(* CoDeSys 2.3 project: cy-wg-017-002.pro *)
(* Title: cy-wg-06 - ClevergyAS *)
(* Author: Andrea Ravasio *)
(* Libraries: Standard.lib 2.12.10 13:48:34, Util.lib 26.9.14 09:12:46, Visual.lib 2.12.10 13:48:34, WagoLibIdent.lib 25.2.13 10:12:16, WagoLibStatus.lib 2.12.10 13:48:32, SysLibFile.lib 2.12.10 13:48:34, SysLibRtc.lib 2.12.10 13:48:32, SysLibSockets.lib 10.2.11 08:20:54, SysLibEvent.lib 2.12.10 13:48:34, SysLibPlcCtrl.lib 2.12.10 13:48:32, SysLibCallback.lib 2.12.10 13:48:32, mod_com.lib 2.12.10 13:48:32, SerComm.lib 31.5.11 07:54:36, Serial_Interface_01.lib 22.4.13 11:50:14, Modb_l05.lib 13.5.15 09:30:08, Ethernet.lib 2.12.10 13:48:32, MBus_03.lib 9.2.13 16:51:58, WagoLibModbus_IP_01.lib 24.7.13 14:05:58, WagoLibMBX_01.lib 20.3.12 15:32:40, LON_01.lib 28.9.12 13:05:10 *)

(* PLC configuration (modules and I/O channels)
VPN_ST2 AT %IX30.0 [BOOLOnX_I] Ch_1 Digital input
LAMP_AL AT %QX18.0 [BOOLOnX_Q] Ch_1 Digital output
KEY_QE_ST AT %IX30.1 [BOOLOnX_I] Ch_2 Digital input
CIR02_EN AT %QX18.1 [BOOLOnX_Q] Ch_2 Digital output
CTL01_ST AT %IX30.2 [BOOLOnX_I] Ch_3 Digital input
CIR01_EN AT %QX18.2 [BOOLOnX_Q] Ch_3 Digital output
CTL02_ST AT %IX30.3 [BOOLOnX_I] Ch_4 Digital input
AT %QX18.3 [BOOLOnX_Q] Ch_4 Digital output
CIRD01_A_AL AT %IX30.4 [BOOLOnX_I] Ch_5 Digital input
AT %QX18.4 [BOOLOnX_Q] Ch_5 Digital output
CIRD01_A_AUTO AT %IX30.5 [BOOLOnX_I] Ch_6 Digital input
AT %QX18.5 [BOOLOnX_Q] Ch_6 Digital output
CIRD01_B_AL AT %IX30.6 [BOOLOnX_I] Ch_7 Digital input
AT %QX18.6 [BOOLOnX_Q] Ch_7 Digital output
CIRD01_B_AUTO AT %IX30.7 [BOOLOnX_I] Ch_8 Digital input
AT %QX18.7 [BOOLOnX_Q] Ch_8 Digital output
CIRD02_A_AL AT %IX30.8 [BOOLOnX_I] I 1: Digital Input
CIR03_AL AT %IX30.9 [BOOLOnX_I] I 2: Digital Input
CIRD02_A_AUTO AT %IX30.10 [BOOLOnX_I] I 3: Digital Input
CIR03_AUTO AT %IX30.11 [BOOLOnX_I] I 4: Digital Input
CIRD02_B_AL AT %IX30.12 [BOOLOnX_I] I 5: Digital Input
CIR02_AL AT %IX30.13 [BOOLOnX_I] I 6: Digital Input
CIRD02_B_AUTO AT %IX30.14 [BOOLOnX_I] I 7: Digital Input
CIR02_ST AT %IX30.15 [BOOLOnX_I] I 8: Digital Input
CIR02_AUTO AT %IX31.0 [BOOLOnX_I] I 1: Digital Input
CIR01_ST AT %IX31.1 [BOOLOnX_I] I 2: Digital Input
CIR01_AL AT %IX31.2 [BOOLOnX_I] I 3: Digital Input
CIR01_AUTO AT %IX31.3 [BOOLOnX_I] I 4: Digital Input
0750-0478 2 AI 0-10V 16 Bit S.E. [Type_8_2_Channels] node 3, in %IB56 out %QB36 {INTTypePAAssignment = PLC; INTTypeModule = plugged}
  VRD04_ST AT %IW0 [WORDOnW_I] I 1: Analog Input
  VRD05_ST AT %IW1 [WORDOnW_I] I 2: Analog Input
0753-0648 LON-FTT [Type_55_1_Channels] node 4, in %IB4 out %QB0 {INTTypePAAssignment = PLC; INTTypeModule = plugged; DataStream = 1F8B0800000000000400ED5D7B6FDACAB6FFFF4AF73BF820DDA3560A0D06421E27CD1605A7419B470E9074576D851C3310EF1A9BE347D29C4F7FD79AB18D8DC70F02348158DAEA26F678CD5A336B7EEB31CBE3F33F7ECD34E18198966AE81F0BE287524120BA628C557DFAB1E0D893A2582BFC71F1BFFF73DE36F4966E1373; DataStream = 222B44808774EBEC97A57E2CDCDBF6FCECF0F0F1F1F1C363E583614E0FCBA59278F857A73D50EEC94C2EAABA65CBBA420AFE53E3F4A70AC2B5694C4D79D682C6A7A5B352E9EC18FE3D3A2B8967A5DA59A90A3F0AC25FEAA42BCFC8C7C217796A8C6E55DBB04D4357954A09C418106DD234146746745BB641BC8631C3DF1F0B; DataStream = F5F15878321C5350D815E19E98C05E9738F0F4A56ACE1E6593DCFA63724A3B1AC80FE45AB6EF3F161A67DF3FABF677E5A958128F8B8F53E15D935844FFAFAC1BC227792ADBB62CD44BE2A7F7DFDBBDEE48278F05A1638C1D8D749DD91D3181620106541070483BB2F9B377F737516C8B5E5BBEEA5E84CB43329B6BB24D5A63; DataStream = E0589DA8C4F4EFC15D1CADD6F8A2541278FF9D1FBAF7034F0C14634E2EE016FB11B8F32779C2EBF8BFC0D5963E26BF2EC4F343F6C3E7EB3081319F699CA58BC1E5F55037C68449B67890DEF41FE1360D37E999EA54D5658DDB3474D37FA465B50DE527195FD8A6434006EFCF40838EAC8F65DB309FFC368B2B8166BD39EA92; DataStream = AC5D4C64CDA2CDFC2B7EAB0EC18966D38D4319FADB6F256904B5AF6138A082B096CE7455FB58C0CE0BC261604088FD68983F6F655395EF3462052765E95EE0569AC63C4F6B9235C7D79ED3F2B2FA0454086F867528558F38BAD4BD1D8E8CBBBF4726F98F43AC386D5A6894FEA0F6BDA6D12621A50936E56A53268D5A41ABB2; DataStream = 6B5654BBC418EDA22DB3691823AAEA03A28F87EA8C4E6DF0CF703BF957A85DE0CFE5767DA210F581049A06AF2C097F6DAA86A9DA4F0BE1FD2BA19603623EA80A193E81E6D5959FBAF1A891F1948C411B0377428F345513900106F2A2A5CF1D98D4C58530CB60F526AA827373D1357460227825D4B461E81375EA98D4AEC02A; DataStream = 9913D35689B53CA82DCBEF6A495996AF871EFBF4649381FA5F7251393FF47F0756FD61FCB27FB58850494284CA261101BC0DDBB132008231705BA6E281DFF2D5C341398783EC70D073ECDDC283DADEE0C171121E1C6F0C0F26AA46D045C8E21E5C42DB3E364D770FFCA61BC4035FD1D301C12399010F8E723CD85FF7402CEF; DataStream = 0F1E5493F0A0BA513CC8EE20E03A47D39FC54558B47DF5A050CB41618F9D84F2F1DEA0C269240DC54688450DA58DA2C2DCC80209D4F45F1B59828645D3570F08C73920ECAF97B06AD010B9B3C838A6B27C7EC8CB5E3F2FA59D9CA02E8A3119EAE28A296ABA286F55D376644D9838BAC2568B70A7C1A02E679E574A2327ACD5; DataStream = 3C8F9C0DFF5F5F1E199A67CD234769673004BE366CD012AC92408AD332DA323705C26BF30D7DF1F28C321BA197CB2843EB8C19E508E51C18F60B185EDE475C1117F627B37C9294493AD95826C906D5C2E53B9B67C10554C401C9E8320449E7C0B05FC0B07B1EC3FE64934E4E9290E16453C8206BB239CB020A75D6300B24B8; DataStream = 347334D82F34D83937A17C9AA3C136D120B38F9003C25E02C2EEB907FB8408491985938D651430E62799F28CDAD380B5CD82082ED91C11F60B1176CF45D81B3C104B492E02BDBB1944B87F9095D1CC18674285AB46431CC12C67CF2704C8E7E8B05FE8B07BFE8298C3C3EF81871C1BDE3836EC9CE7B04FD07094080D471BDB; DataStream = 85802BA34C3B101417B059F66D0897768E0BFB850BBBE733EC5348F17A81214785B78C0A3BE72DE4A0B06D501838F3790E0C6F1D187277214F31B883B40087729E81CCE16147E1619FD20CAF1A1E726C78E3D8B07331C53E41C36B8C29CA790632C7855DF419F629A478BDC090A3C25B46859DF3167250D83628E419C81C18; DataStream = 7277214F31F883B400874A9E81CCE16147E1619FD20CAF1A1E726C78E3D8B07331C53E41C36B8C292A790632C7855DF419F629A478BDC090A3C25B46859DF3167250D83628E419C81C187277214F31F883E48243F3EA4B9E80CCD16147D121CF326CD16F4068A82B76EE35BC755CC8C3891C16C2B000DEC2B5A1EA79F2F14D; DataStream = E3C2EEF90B39306C1918F24D891C17727FE1E560E13409154E37060AD6A36A2BF75940A171D9446F41D27194321E00E912CF6161BF60217717725C08E1C2E71C17725CC8DD857C4FC21BA4B0CF90173EE6E0B0834E43BE27B1C51C034243BE21F1D64121F718724C88B80BF986C49BC785DD73167260D83E30E4FEC25BC785; DataStream = DC5FC8138F1E287CEA35F20D891C16727741C8714158C2857C4322C785DC5DC83724FC410AFB0CF986440E0E3BE834E41B125BCC312034E40986B70E0AB9C7906342C45DC83724DE3C2EEC9EB39003C3F68121F717DE3A2EECBDBF10B9632D6EA5F17C7ED836F48E6CFEECDDFD0DACD1AB4BD7AC8BF37F7C6B34EBC3FAB7F3; DataStream = 3F7ECD34E181981650FB58103F940A02D11518307DFAB1E0D893A2582BFC7171DE906D5933A617E797AA46849605FFB38949C6F0484168C2CD5B9F44156960339CC28F05FC17FE36CC996CFB8D6AD8A623FF6D9881E70AC2B56CDF7F2C34CEBE236A99F28C92B18477BF4E6AEFBF83085F6048ACEF48D1FA3E18D6BBCD7ABF; DataStream = F961F8F51A9EA430F7B110838305A14F26C0AFAE90C456A8D2035B9ECD819FF2A158392C97C4B2209E9C954B6762B970B18CD69415EE55E1936CB923308095AAD8DF6A3F0A025DC2207E41A0E0F9B1705C2908084B1F0B74604DF21F8758365C7BB0D9C3886320A1341A0CFB378D2193148606465355D89314EB26F0F8081E; DataStream = 2F08A865C87E41B8D155E8EC9F9AFDAF96FE206BEA58B06C132616BAB10CC754C83FA7F6BFF84205D89774672678E491BB918D73F74B9D39332A0A800CFB5D143D61FAF17248DD9B0E4F0A5FF4813AD55DC57245F12499048648D0E129AB202077842D0677488F10145364BAD12DDA0BE8D414E6C26AE936991293F6D5B206; DataStream = 8AACC9EC8F859C474795234F3CDA134FB89BEEA0F5B92B3547ED5EF77341E84D2616B129A1A8C02A23829D917A40DC72485CB7D5B62572215DB06101180E77E26264ABF02793921BF9E4E2A59CA99AA65A4431F4B195494E98E96F95C55AF2175013B402AC3C6A82208FC7A0E3165F8C56AFBB60FF88C7FE18B5DCA7C1183E; DataStream = F218F670C8EF24E3FA2F2F782E7B3CD71909C1C6C700786DF32969ED27328DECD81EB7158F5B5E0F597569706F20C52CCA54A90470A05289C8478D40824E0DAE7AFD340119918826F9F07052BC536DC171991700F19883B4DD95131E60754564A83D0B19C45A9CA8CB8E0375A39E639F5CD3E2DCE9C42EEAC69824ADA94CFA; DataStream = 69E9F14BC9E2F4B3052D15034A2AEE928E7E526D7F72960472C1CF98C9AACE63FF536B7899A26F63F7E178B6FD89624D57B64AC2B14045807F0236D115E8382850F9D813A90BCAF04C8174FA68BC3854CF741A69AD2244352244D517A21A14226056016F05059BA48B72CCB7A4D42624C842C5108C89804D5592CD883E5BA2; DataStream = A129EB964C431EEA2C98E9729D7017CAAF91FB78BC68B4018C1E4CD6AA60BE0228948F8EC270B70A089C7291CE25132F196B1154C13580FBF847702931163E9B86335F1BB2A7F378C89E867A581BC0D25038AC52CFC2DE3BC3D088AC6F03B66A0B15823E9FC9BF451FCD00C26CE859F3376F3A181F37BA6341DB894AB4F133; DataStream = 457128892451D222E9DC94E4A62404C06B5B9229A3B29E4AF24DCB730CCEF35C6E17E01DFB1EF7041416A11B5CC4891B1CB1C48D7881E4C848449FD531FF39B27939EE55A5E2E685E6406C05A9D6701CAA3F822BD4CB4856431949CB966D27D183484A487A4FBBF1EBF1E67392AC87504A5214B939C941AC247129C905F789; DataStream = 1949D62C3E2159DB7E12A2EB2337721493F7CA9E9A648660644C462EB9F854846B90B62DE0806844B1A985D792A3F40CD949CB253662C4369681C5CC644296EFB9D948796CFA9C6D2CABEF42404C225531D5B96D700D72A6C0611C20B169CEEBA6293F7D136B3F50DD2FD90C4D0C41C6CB02615BA50B8F17B75A2CFA4800AF; DataStream = FDA77802D6FBFDFAD714F928F430022E22D43CF1181FC09A5813947BD9040787981992C4747534E0818CB607C1348072E5938870CB43C2994BB6641A57F5FE42E032D7D6FA127F138F7E2CAD99387464C9AEFAA0D16A2D86E2F9468BF6F36F471E6774C6C4EA71F5A452AB1EA7C566EE30FCFBA6DE0C0C0317193931DA92F4; DataStream = 55DF483FD92B79D0CF44C6615ADA320C88E55542E7CC6B76A38E482A6866DE0E096CDF9C6E167E18FAB0D059683563D0870B3EFE43CF051F16488FD4B1275B147B6A02D3BEEDC638B1E2AFEBD8FB127E8B604DB66CFA6F0A6E6A4B23A1117D6ADFAF1F02B8F27BE4E20740EA0A62F5B4745214BDF48AF7CCABCB946241C266; DataStream = 52A59B8FE3D2371D62A5E23A98ABEE3FAC12A1AF01B362608B4F5CD4A09C54822112111EC0394EF6FD62423E0C840867B3125D68F5411D3BB226E082A5EB74033963C62E522CC5A78EA2BCC203A5CDE40CE2139329FC8A2BF22B6E87DF72567ECB2BF25BDE0EBF95ACFC5656E4B7B21D7EAB59F9ADAEC86F753BFC1E65E5F7; DataStream = 68457E8FB6C36F2D2BBFB515F9AD6D87DFE3ACFC1EAFC8EFF106F9CDC6E1497AB29EEBDAC0B3272F0CBEA7CF67FDF48571584C307469BC8B5B327A9941594CB07AA9CC6FC90266466831C104A632BF25739819AEC5047B98CAFC966C6366EC16138C632AF35B329499815C4CB094A9CC67B69A1BABFAF322023F0B8305F1B8; DataStream = C131E3EE65A6C403B8E93A721F66DCFB1B404F44360F8499A1DBF707C2587E3A10EE0D07AFA8BA63930381150467CC9A66CF9C554A58E5CFD91CFA4A647EC413CCA145C57CA28F25A503CB4189574907AE14BF7A6274704057895FB941F98C5189D73DDA604BC254168932995B0C1D270A37121FCB89150F707B4B6294FDA0; DataStream = FA0A147B1539AA3C39EE29917841F0FE9624393AF5B58B2ECEB56B64672E9904FDA22DB62ECF8081CC0AF2700B875CAC4ACA61055E6F58277F13C8938B8B1DFB137FEBA70EC2CE9EBF658F6335F3816B2B19F3B6E1D67FAC9030F79E49C8974705D2FC875E36471E27F09A6BC8136FB504390ABC767EFC99FB54ECD5C3986D; DataStream = 8F55DE8E302821B6FD11BB61C51A65DEBBA7F52454FD47B815162A27A994431E4325BCD8EC98ED3756539258B7B6E82F691355F6BB89AF3039CE2AE2DC2D541A69E4816859AA66FCD226FA44BAA4DC32B670B749D2CE43DDC54B7CF29B5EF243A0E8DEAE524FC3DDD0A27A38B28D11E26C92DEAA8B4E0545762C045B179653; DataStream = E565385BA5387B8B29F61890ADF240F696ED9DA5EE48F2B771DC9DB7A51D701F6AABBF056AB932AFB095C3055A2A192D934908C57E2FACB22026396E89D34E2EA272A2981D085D442EA8EE66EC227261730783177EF1D08E462FFC12A01D0E5FCAFC3DF895E2974DA3D9E9696086FC57C157A968E206FEB320AD8DBD7D1E34; DataStream = B1CCFFD3D41978D82B18DAC06319CC2DBF5C8B798E2E8D9735BA09A3B0825E26F8C794F47A06788D903B5CCEEB3A9FA7BEF9A5B59673C352E3E2D32C45F2F07C244A9DE3E967C43CF0EA79B65F1CD927F2F8F00BF8DE2810ED3CB55492F38AD1E3686EA764447D4DA5D5D538758BF714B77FCC852F64865AAD30CE70F37220; DataStream = 706C95960F328BF7AA1635A11BD749DF917203EDE71F2503B1F328701A4BE8388956F3C0A7FC8A1206BF314BE012E69D8553AE7243E8F4090987D05C231DEE3629843642DDC587D018A9AEA98881CDA3F262F7E8B4B224F9B31392A889E157886A4145745FBC9968F234BB99DB1B6D4C2DD67073B6C556930E51FA462457F1; DataStream = 544685CFFB06B652C56C4278EABC0149166BE8F7977234550B898CD79163ECD27891728E9E63178D49917A65D63A52188E8D2F9831422F52DCD19B13BDA8A8A6E2A86BE9950174462E9D1729F470E7C46227276E60525C4A2F52F8D121CABDACABD07171223BDA5A3333F3698D28AD172906B924647C272B3F411C5573CCB5; DataStream = E667E2D21AB9B47E53D95FEF81984553D6A75999E786E4065019512A2F62496EC0AE6E400A07C96C538C140B22E1BBABE6CAEB832B0BF1696D737DA458941BFACDA0A26D146744B6B22F9098D94162B8D3E2127B11CBD230663347778F3AB0565CF85CB914A0B885459FDDC65C42DF640C36469B14EDEC8E18571894638494; DataStream = 46F6D6FCB0B4F2424F8EA2AA17E7C8211E3EB4864CBE3823551F79045FC4DEB093888B60CAD79147A35446FCC33BB761633AB2EE00A629866E9B869691756E4E6646298D5C4A2F14B5CCC127635BF76B4802AAE4D5E4FC7E43C36440A36DAAE3ACE015278647E6452C4C9FCC0DD32ECE64EBE73A629894CC08C9BC8855F138; DataStream = 52F56911BF8EB58E2CF3052DFAA5AD17B1294181D0266C4A20A4F52256856E861475C356274FC5F16AA13E572AB605C2088EB61BF7A758953EB1F8EFFB665A38700FF07836D748F2CEE9338EE83B1182A6C52F85C43ECD0732CEF0DA06778B2DF0FC364EDF5A23D1BF78079B7E40F3196955CB7D7029FF484B5D5856956C65; DataStream = D77051B6125B6DB4BC43185F6AE44E8AF78EC42796715F9AA0FFA34722399AE695AFA5EAD5609D3385C3874D259D35B25CFF1177FC54CA6123BEA0B42D3DDF6ECDF355DCF4B8B7457094B1F0A57C5C0B9D47533EAE88FED6227EB105F71E68ECB2F23B16814FB98407C39BF672D26B1763029E38B18406D12CD5C9B2C54877; DataStream = 79E82728EDC0409C8414993BE757B7F586308B394020EE8CB1F0072F93A6D8279FB0A5538D9D7DEBE23CD03EFC97B0F872C2509EBA67FD2C36B82ECE59655D28212FB84B382AD1657FD4BD691784BEFC48DBB0213A0C53192075DD56654D901505632F93E0DE35975CEF5AEA8E86BDD140EA3633507AC4FDDD14527DA921B5; DataStream = 6EA5209751261B9A611141D601DCE507E21E3DC625DB68F706D2E8B2D50E512C27501C13B485E9349B525B1A46495722A4FBF4C84E60734C3F4963984FDEF704B8D49B2D188261AFFF15D65DEFCF9BEB20F16A9438B06CCC569CAA51BF1EA47A94427585695BA2CC0ED83B0C683457BD6B41F5F6CF0D5C55BB0719B49B9685; DataStream = D878BCE9849882E55001C10CC510FCEB520211FF8C9069FA33A919C64F3CF2378D129B4B4A2B49B125D3344C014FE19C131DBD9658351CB0A1BFACB7DAC99AED931C2F319DCCA9D4EF27AB757828555D58E456E2C7F2A6DB94FA5FB08E2A49A97D96519F61140E51035346A3D55B6639AAD66196F125C8B140F3285C8AC356; DataStream = 47EADD0C97C9D62264BFA8B05A1E058BE29D420482ECC710FDD2EA367B5F96691E47682E1DCAEA2718B944EB37C3AB65922751926C35334365D8A0B3730C9B091F31806AA3210D063065F5DB25253B4D018C3BF26400924A3DEEA908407A20497F8E5ADDDB7A1BB7ED030BA2149D33B7F5977A8BEB7586EF074889D9B0E7D8; DataStream = C59ED03B2661166EE663F4E1FCF9BD07AD24DC09AEB74757521D543C0C43D1C5B34C726218762CC9CB5E6FB84C32BACE9BE4CE99D2E305F1835E28E13B9C655967AF29BC8F21DE943EDD7C0ED38EC2522B40D561AC6722DEEA5EF6C2B4A3133C78B2C0875C9DF1C1D7C150EA44BB88AECFE1BD7BB6B4A05A825B6B10431434; DataStream = F246E26966318A2621B232B8F83A982EDD3D44299B0C8D5E17BF961652DC62140FB1A731A15BC8D095319968AACEC50220D9BBBC6CB7BA2197A418D53F561C8AC5B52A9B541DBFF407233F939F60F90A6368691B54AAC08689074302A0F3BD6C8E1F65DC3B61D7E244BCE9FED9ED7DE986F8892AAF67DD03EF54B9C3282F71; DataStream = 4A916B4E14FC84E538AED37447A06B08CB94E79859D0B9D60049F670B69AAD213D16767939EB3E4B2B92ADB73B41BA49BEC1D0B065EDD0AB25A085A00FE85BD3FE44E11DA6710C1DBAA2156660EC2DC16B0CF38567D0D94497016DE2466DD81B8E06B70DCA9398EC5424F2C2DD205FA25F4E762E12E973B74596E857923D0C; DataStream = B7381AACB65B20CD264D23B22970437E20DF06BBDDEE0CC1FDEF8787270A0D49E4E3462748BE9CEC7030F2F7EAF47E05F6AF5A9FAFF8FC73BC8FA40EE2040875504EF145B8039436F211C58C3A227CC269631ED1488E9D8A1993D4E18E30CDB1AF31B453473ACA7774A95E02122C83529CA3D1EA23C910419EE30F0401D58A; DataStream = D9895EF7A508E1E8A244C24593E0B786C7E0A61BCE1DB8EBEF68FDC3FB4CDD0CFB9F42B82FF24280401FE00123C25806FD7E8707D8EFC887E987033032A6AAFFD420504004B7124C1C763DB8B9BE0D751D5DB561F170879BBAE2D94771280D8691618C2EDE987E569B31DA176FDAA26B39D4DF8CA5E204A23FA8A6A1E3FB26; DataStream = 80DB689A886E312782BD400CA19D72CF8F3D5C16A4EE6DA3D7B91E75EA7F8538882EFA1007F29D8E8EA4065663EED89984EDF4BAAD61AF4F0D71C8EE71C291B0B0BE4D856924669C91A77DD45B5D9C3DA91FF2F6CA9C1C057ED15790E773CD73BB62034AA45D1FC2BF10FCF5C2F17A94F51E449426A3953A2A517A513E193D; DataStream = F00169A2228DE2977ABFDBEA86228D4A395B8876E286689177E457CC105D67C97FB68D472CA2612B65BEF48E3D97665BBA95DAA3E878FBB7B826227837C9EBF3DB718D41F06E92BF7605A6E559625592FDB4B63A21C2409E102046ED02B56496F0EE53BD818703FB871494B9E079BDE489446DC235FB8EF653A64E2A719D94; DataStream = 93DD354A74103006CC1E47E857E3E85792FD354A7FC80CDAE125AD0D7CD754ADB9263FBD8FF67214D74B35D969A3BD5C033C51EE0F04BA2DD1C0CC9902782241483047388E13AE16D76D2DD995A3DDC4CDC8491CD19364372E8EF7FEB07BC074007E250DA2588A55B8528AA347FBA6E4358605DE72E175133B6A628DE3F3A5; DataStream = 421DB243B12EF232D38A58D7FF7706AC93684DA6FBE214DDFC30C9CC78802B7E51109F72AFDFA9B73959712B402FE6D9666B50FFD4969AC9A8C70A833CCEBC378DB8046FAE9BF521EEACD78737836414BC262626997CB25EA9610CE581D4BEA48E503206BAB93C3974C45312ABF576BDDF49863D577EF73D2A3C2A88153771; DataStream = C9F6A5EB5E7F081EC6E0CF649CEB7925638933D4BB05EBDF6A4AC99816D29D184A5217A73A19B5FAAEC6B1294951BC7EE796CB5E14951A3454CDA23F8DB654EF73D4270A4A219A6EF95F02C9C83473B0C61D45A63BB49A48F54EC7E252A63461FD0D5B975FDDE16D727086B72A9FD70777B9723699424832A1F926ACF514FC; DataStream = 5A4F6E579D7AF706D3A0C37E386E8B2EB268070855B4B222A983BED4E9C18A8B74C0D973621D04AAD5B04285A6F598181375EAB8603D674E09FD0E23B7DBEB7EEF73BF1E9EFCE87264FA446BB08A5E0D16AD4913DE850BB3B836C6D7B3BE3490C25B1F9CD5FA8B280E50679DF9DB0E2061E2028E928E2E60260540A02C68C6; DataStream = 3491D3762FE4FF7362C9B62143CC7AEFCFC322D58B3B8C83C6F5106FB06F8EC574D5EED59BDC09E0EC5A393AED4C714C13BC0B0D7746E531F4E5F6FE41684D42DC3CCA96702F6B2CF643FDD69E0EA0816A098FAA8631AD05165D301D9DEDDD9AC68C3D8EAFED63EA7EF1FC87B811BFE9F298E744A257402785FBA1CFD9DCAD; DataStream = 9A0B8F2D2D4D42B32FE377DE9956808F05A382697FBC11142BF82815ED11E23F22806D4A17EBAADE1E72E5E2997EE0CB4C166D31B47764AAD2D18E1D50B0DFF53EBFF3288EDDE89AA781717DC7D9F66E9CE2953968C696A3453BD2C92F1B970E75758DB9E711BEC34D1EB7E80F7DDF035801162D3F84BB07EC01E10EDF0638; DataStream = 1088AD7C788FAB394D1F96277FE6807F7B47847FFEC731EC7FA9638DB05FB863C07EB17975AFE29690A290B9CD94DED59203C1C054C0A36A316D409D019AEA54374C508950B726B11D53B7901287BEAB91131B1315748CE8174927A1EEE2BCB5A174CD1DFE6A46D7BBEABADE6E8519DFE17E8873B8316AC8E0723798B9C2B4; DataStream = A2ECD806258030829F61D3A704F7CEED4742F450FE07F3775C53433BADDF0C7B51742032AD9830748D5B68449FBC92EAC3643FBCBEE0A2E842B102ECB094CF23D654F3EB4828F94EBFFB79F4A5DF09D730716AAF0C434BE5B5D1EBB593FD702EAFBA3ABD8708CE31A709B3D6FA7C050071D3FF2C257BE5DC1E30AFAA187C0F; DataStream = 8492C72CEA32F71C6760A118B8C5E9BA356C5C1C7BEED8F10AD0BBBC4CF1D5FDF8F98E20418C79F8A9574A6F39E489DA7C0916CF143C8827AC85B05949C93BFA73EECCE65C778552963A52FF7344ED38DB43AA3F0A2CA94800642632586B000F2CDAE1FAAEB48BCB7A77D4EBB6BFA6B8F2AECA3DAAF63DCD4E638ADF609DBA; DataStream = E63BBE87BE149D508E6FDF52487126FFC46E5805690CBD56434A71E1DDFA563AD8A9E43AF5BFA20B9BE3B1C3D81A33D05F448A431C8F64B252A3D7ED75BEA6B8E94D72EFCCD4B11F6224D36C4A57379DA50AA0E8AA6B00F0DE9919C835EAEDD6A73E44D8297EF7427B9574B1A9C646669BB3C67CA2B0B6C0D065A00A16AB9E; DataStream = B699E34F29632161CE233CF25375A3ABDB06F591E3AD82DF20D17966D0D94BA6E5DF8FB8B2617B7C182E813EC44ABD8B735AAFD7B2E07FE010B8B5D74D08346E89694143D4960F400D9BB1A2EECB39440597B48EC86F73844D3AF2DF8619780C1896ED7BD0ADB3EF2EE7948A25BCFB75527BFFBD6DE85F0CF3A7F59D16687F; DataStream = C71A9D66BDDFFC7079EDD6A0B580995249E0FD07B29209B00BF155622BFC80C3003FC180CBF350AC1C964B6259104FCECAA53358AF20BDA3535F4FD6A047FAB967CE35DF7BF16ADDF13B7942CF0FEA545D51E7B216736AC10004C24FDEB9ED2305F830F81DF0B864AC1A65EF15103C308B7DD43AD0E9F2414AD19EF407B5EF; DataStream = DDC5410D1C8E15ADFB4FE976F940ADF8F48EFE60781F170F765AE1761AEEC47F99872A61B264D804A40B75729CA5935AA8934439B005CA12EEA49AA193E350278B33F16245B93696C6CB5DB111E5E35D5BACDEC3066E641AD38B1F3FE08F36BE0B01CB78222BE4E2FF01E50CEFEAD6460100; DataStream = .; DataStream = .; DataStream = .; DataStream = .; DataStream = .; DataStream = .; DataStream = .; DataStream = .; DataStream = .; DataStream = .; DataStream = .; DataStream = .; DataStream = .; DataStream = .; DataStream = .; DataStream = .; DataStream = .; DataStream = .; DataStream = .; DataStream = .; DataStream = .; DataStream = .; DataStream = .; DataStream = .; DataStream = .; DataStream = .; DataStream = .; DataStream = .; DataStream = .; DataStream = .; DataStream = .; DataStream = .; DataStream = .; DataStream = .; DataStream = .; DataStream = .; DataStream = .; DataStream = .; DataStream = .; DataStream = .; DataStream = .; DataStream = .; DataStream = .; DataStream = .; DataStream = .; DataStream = .; DataStream = .; DataStream = .; DataStream = .; DataStream = .; DataStream = .; DataStream = .; DataStream = .; DataStream = .; DataStream = .; DataStream = .; DataStream = .; DataStream = .; DataStream = .; DataStream = .; DataStream = .; DataStream = .; DataStream = .; DataStream = .; DataStream = .; DataStream = .; DataStream = .; DataStream = .; DataStream = .; DataStream = .; DataStream = .; DataStream = .; DataStream = .; DataStream = .; DataStream = .; DataStream = .; DataStream = .; DataStream = .; DataStream = .; DataStream = .; DataStream = .; DataStream = .; DataStream = .; DataStream = .; DataStream = .; DataStream = .; DataStream = .; DataStream = .; DataStream = .; DataStream = .; DataStream = .; DataStream = .; DataStream = .; DataStream = .; DataStream = .; DataStream = .; DataStream = .; DataStream = .; DataStream = .; DataStream = .; DataStream = .; DataStream = .; DataStream = .; DataStream = .; DataStream = .; DataStream = .; DataStream = .; DataStream = .; DataStream = .; DataStream = .; DataStream = .; DataStream = .; DataStream = .; DataStream = .; DataStream = .; DataStream = .; DataStream = .; DataStream = .; DataStream = .; DataStream = .; DataStream = .; DataStream = .; DataStream = .; DataStream = .; DataStream = .; DataStream = .; DataStream = .; DataStream = .; DataStream = .; DataStream = .; DataStream = .; DataStream = .; DataStream = .; DataStream = .; DataStream = .; DataStream = .; DataStream = .; DataStream = .}
  AT %IB4 [BYTEOnB_I] First Byte of 24
  AT %QB0 [BYTEOnB_Q] First Byte of 24
0750-0464#04 2/4 AI RTD / ADJ./ HA [Type_44_4_Channels] node 5, in %IB60 out %QB36 {INTTypePAAssignment = PLC; INTTypeModule = plugged}
  S01 AT %IW14 [INTOnW_I] Channel 1
  S02 AT %IW15 [INTOnW_I] Channel 2
  S03 AT %IW16 [INTOnW_I] Channel 3
  S04 AT %IW17 [INTOnW_I] Channel 4
0750-0464#04 2/4 AI RTD / ADJ./ HA [Type_44_4_Channels] node 6, in %IB84 out %QB60 {INTTypePAAssignment = PLC; INTTypeModule = plugged}
  S05 AT %IW18 [INTOnW_I] Channel 1
  S07 AT %IW19 [INTOnW_I] Channel 2
  S06 AT %IW20 [INTOnW_I] Channel 3
  S08 AT %IW21 [INTOnW_I] Channel 4
VRD04_CTRL AT %QW12 [WORDOnW_Q] O 1: Analog Output
VRD05_CTRL AT %QW13 [WORDOnW_Q] O 2: Analog Output
0750-0650/0003-0000#03 RS 232 C Interface (Adjustable), 3 Byte [Type_21_1_Channels] node 8, in %IB100 out %QB60 {INTTypePAAssignment = PLC; INTTypeModule = plugged}
  AT %IX22.0 [BOOLOnX_I] Transmission acknowledgement
  AT %IX22.1 [BOOLOnX_I] Reception request
  AT %IX22.2 [BOOLOnX_I] Initialization acknowledgement
  AT %IX22.3 [BOOLOnX_I] Input buffer is full
  AT %IX22.4 [BOOLOnX_I] Number of received characters Bit 0
  AT %IX22.5 [BOOLOnX_I] Number of received characters Bit 1
  AT %IX22.6 [BOOLOnX_I] Number of received characters Bit 2
  AT %IB45 [BYTEOnB_I] Input data Byte 0
  AT %IB46 [BYTEOnB_I] Input data Byte 1
  AT %IB47 [BYTEOnB_I] Input data Byte 2
  AT %QX14.0 [BOOLOnX_Q] Transmission request
  AT %QX14.1 [BOOLOnX_Q] Reception acknowledgement
  AT %QX14.2 [BOOLOnX_Q] Initialization request
  AT %QX14.4 [BOOLOnX_Q] Number of characters Bit 0
  AT %QX14.5 [BOOLOnX_Q] Number of characters Bit 1
  AT %QX14.6 [BOOLOnX_Q] Number of characters Bit 2
  AT %QB29 [BYTEOnB_Q] Output data Byte 0
  AT %QB30 [BYTEOnB_Q] Output data Byte 1
  AT %QB31 [BYTEOnB_Q] Output data Byte 2
0750-0653/0003-0000#03 RS485 Interface (Adjustable), 3 Bytes [Type_21_1_Channels] node 9, in %IB100 out %QB64 {INTTypePAAssignment = PLC; INTTypeModule = plugged}
  AT %IX24.0 [BOOLOnX_I] Transmission acknowledgement
  AT %IX24.1 [BOOLOnX_I] Reception request
  AT %IX24.2 [BOOLOnX_I] Initialization acknowledgement
  AT %IX24.3 [BOOLOnX_I] Input buffer is full
  AT %IX24.4 [BOOLOnX_I] Number of received characters Bit 0
  AT %IX24.5 [BOOLOnX_I] Number of received characters Bit 1
  AT %IX24.6 [BOOLOnX_I] Number of received characters Bit 2
  AT %IB49 [BYTEOnB_I] Input data Byte 0
  AT %IB50 [BYTEOnB_I] Input data Byte 1
  AT %IB51 [BYTEOnB_I] Input data Byte 2
  AT %QX16.0 [BOOLOnX_Q] Transmission request
  AT %QX16.1 [BOOLOnX_Q] Reception acknowledgement
  AT %QX16.2 [BOOLOnX_Q] Initialization request
  AT %QX16.4 [BOOLOnX_Q] Number of characters Bit 0
  AT %QX16.5 [BOOLOnX_Q] Number of characters Bit 1
  AT %QX16.6 [BOOLOnX_Q] Number of characters Bit 2
  AT %QB33 [BYTEOnB_Q] Output data Byte 0
  AT %QB34 [BYTEOnB_Q] Output data Byte 1
  AT %QB35 [BYTEOnB_Q] Output data Byte 2
VRD01_ST AT %IW26 [WORDOnW_I] I 1: Analog Input
VRD02_ST AT %IW27 [WORDOnW_I] I 2: Analog Input
VRD03_ST AT %IW28 [WORDOnW_I] I 1: Analog Input
AT %IW29 [WORDOnW_I] I 2: Analog Input
VRD01_OP AT %QX18.8 [BOOLOnX_Q] O 1: Digital Output
VRD01_CL AT %QX18.9 [BOOLOnX_Q] O 2: Digital Output
VRD02_OP AT %QX18.10 [BOOLOnX_Q] O 1: Digital Output
VRD02_CL AT %QX18.11 [BOOLOnX_Q] O 2: Digital Output
VRD03_OP AT %QX18.12 [BOOLOnX_Q] O 1: Digital Output
VRD03_CL AT %QX18.13 [BOOLOnX_Q] O 2: Digital Output
Fieldbus variables [FB_VARS] node 1, in %IB0 out %QB0
Flag variables [FLAG_VARS] node 2, in %IB0 out %QB0
Modbus-Master [MB_MASTER] node 3, in %IB0 out %QB0
*)

(* Global variable list: Global_Constants *)
VAR_GLOBAL CONSTANT

	Plant_NAME			: STRING :='cySN:17 cyVER:1 - ';
	Plant_SN			: DWORD  :=17;	(* S/N Impianto di telecontrollo *)
	Plant_SW_VER		: WORD   :=1;		(* Versione SW installata *)


	(* Colour defines *)
	COLOR_RED			: DWORD	:= 16#2020F0;
	COLOR_YELLOW		: DWORD	:= 16#20F0F0;
	COLOR_GREEN			: DWORD	:= 16#20F020;
	COLOR_LIGHT_GREEN	: DWORD := 16#006000;

	(* Parameters *)
	Plant_DefaultTAmb	: INT	:=100;		(* [.1°C] Temperatura ambiente di default in caso di rottura sonda *)
	Plant_MaxRunTAmb	: INT   :=250; 		(* [.1°C] Temperatura ambiente massima funzionamento impianto *)
	Plant_AntiFreezeTAmb: INT   :=-40;		(* [.1°C] Antifreeze temperature, start circulators *)
	Plant_VRD_TAlarm	: INT   :=850; 		(* [.1°C] Temperatura di allarme VRD, blocco *)
	Plant_VRD_TMax		: INT   :=900; 		(* [.1°C] Setpoint massimo per uscita VRD *)
	Plant_VRD_TDefault	: INT	:=300;		(* [.1°C] Temperatura di default in caso di errore climatica *)
	Plant_CirOffDelay	: TIME	:=T#30m;	(* (Def.T#15m) Ritardo spegnimento pompe per ricircolo caldaia *)
	Plant_CirOnDelay	: TIME	:=T#15m;
	Plant_MaxWaterLoss	: WORD  :=2;		(* [lt/h] Massima perdita del circuito *)

	(* Filesystem *)
	FilesPath  			: STRING :='S:\';

	(* TCP Logger *)
	Logger_SERVER		: STRING:='';
	Logger_IP			: STRING:='192.168.100.3';
	Logger_PORT			: WORD  :=80;
	Logger_GETSTART		: STRING:='GET /cygmsrv/hsgm.ashx?';
	Logger_GETEND		: STRING:='$R$N$R$N';
	Logger_CHECK		: STRING:='True';
	Logger_CRLF			: STRING:='$R$N';
	Logger_DataFile		: STRING:='S:\LOG.DAT';
	Logger_DataFileOld	: STRING:='S:\LOG.BCK';
	Logger_IndexFile	: STRING:='S:\LOG.IDX';
	Logger_ConnRetries	: BYTE:=5;
	Logger_RecoverMsgs	: BYTE:=25;

	(* TCP Remote *)
	Remote_PORT			: WORD  :=10;
	Remote_WELCOME		: STRING:='Connected$R$N';
	Remote_OK			: STRING:='OK$R$N';
	Remote_ERROR		: STRING:='ERROR$R$N';

	(* TCP Sockets *)
	MAX_SEND_TCP_SERVER					 : DWORD:=3000;(*60000*)
	MAX_RECEIVE_TCP_SERVER				 : DWORD:=3000;
	MAX_RECEIVE_TCP_SERVER_SOCKET	 	 : DWORD:=1500;
	MAX_SEND_TCP_CLIENT					 : DWORD:=3000;(*15000*)
	MAX_RECEIVE_TCP_CLIENT				 : DWORD:=1500;
	MAX_RECEIVE_TCP_CLIENT_SOCKET		 : DWORD:=1500;
	MAX_RECEIVE_UDP_SERVER				 : INT  :=1472;
	MAX_RECEIVE_UDP_CLIENT				 : INT  :=1472;
	CONNECT_WATCHDOG_TIME				 : TIME :=t#10s;

END_VAR

VAR_GLOBAL
	TestNodoInterogato: BYTE;
	NodoDaInterrogare: BYTE;
	InibiscoModbus: BOOL;
END_VAR

(* Global variable list: Global_Retain *)
VAR_GLOBAL RETAIN PERSISTENT
	Mode_Manual : BOOL := FALSE;

	GRU01_Clima	: typ_Clima;

	VRD01_Clima : typ_Clima;
	VRD02_Clima : typ_Clima;
	VRD03_Clima : typ_Clima;
	VRD04_Clima : typ_Clima;
	VRD05_Clima : typ_Clima;

	Ctl01_Counter	:	DWORD;
	Ctl02_Counter	:	DWORD;

(* Impostazioni di imipanto *)

	DelayAllarmeTemperaturaNonRaggiunta: INT;
	DeltaInterventoAllarmeTempeaturaNonRaggiuta: INT;
	OffsetSetPointManuale:INT;							(* Offset al Setpoint manuale per comensare lo scambiatore *)

	SogliaMinStartAntigelo: INT;
	SogliaMinStopAntigelo: INT;
	BitAbilitaAntigelo: BOOL:=TRUE;


END_VAR

(* Global variable list: Global_Variables *)
VAR_GLOBAL

	SYS    : typ_SYS;
	Logger : typ_Logger;

	Lamp	:	LAMP_AL_GENERALE;
	T_AMB	:	INT;		(* Environment temperature *)

	(**** PLANT OBJECTS ****)
	(*...*)
	GRU01	:	obj_CAL_VT300GW2 := (ID:=1);

	(* Water counter - 2 PULSES/LITER *)
	CTL01	:	obj_CTL	:= (ID:=1, Peso:=1);
	CTL02	:	obj_CTL	:= (ID:=2, Peso:=1);

	(* Heat counter *)
	CTB01	:	obj_MBUS_CTB_SHARKY775 := (ID:=1, Address:=16#49858612);
	CTB02	:	obj_MBUS_CTB_SHARKY775 := (ID:=2, Address:=16#51867882);

	(* Cronothermostat *)
	THER01	:	obj_CRONTER := (ID:=1, Local_MaxRunTAmb:=250,Histeresys:=10);
	THER02	:	obj_CRONTER := (ID:=2, Local_MaxRunTAmb:=250,Histeresys:=10);
	THER03	:	obj_CRONTER := (ID:=3, Local_MaxRunTAmb:=250,Histeresys:=10);
	THER04	:	obj_CRONTER := (ID:=4, Local_MaxRunTAmb:=250,Histeresys:=10);
	THER05	:	obj_CRONTER := (ID:=5, Local_MaxRunTAmb:=250,Histeresys:=10);
	THER250	:	obj_CRONTER := (ID:=250, Local_MaxRunTAmb:=250,Histeresys:=10);

	CronEd	: 	obj_CRON_EDITOR;

	(* Pump *)
	CIR01	:	obj_CIR	:= (ID:=1, OnDelay:=T#1m, OffDelay:=T#30m);
	CIR02	:	obj_CIR	:= (ID:=2, OnDelay:=T#1m, OffDelay:=T#30m);

	(* ModBus Pumps *)
	CIR03	:	obj_MODBUS_CIR_DAB := (ID:=1, Address:=1, OnDelay:=T#1m, OffDelay:=T#30m);

	(* Modbus double pumps *)
	CIRD01	:	obj_MODBUS_CIR_DOPPIO_DAB := (ID:=1, Address1:=2, Address2:=3, OnDelay:=T#1m, Mode:=1);
	CIRD02	:	obj_MODBUS_CIR_DOPPIO_DAB := (ID:=2, Address1:=4, Address2:=5, OnDelay:=T#1m, Mode:=1);

	(* Valves *)
	VRD01	:	obj_VRD_POT_new	:= (ID:=1, fFeedback:=FALSE,Local_VRD_TAlarm:=850);
	VRD02	:	obj_VRD_POT_new	:= (ID:=2, fFeedback:=FALSE,Local_VRD_TAlarm:=850);
	VRD03	:	obj_VRD_POT_new	:= (ID:=3, fFeedback:=FALSE,Local_VRD_TAlarm:=850);

	VRD04	:	obj_VRD_new 	:= (ID:=4, fFeedback:=TRUE, ReducedRange := FALSE,Local_VRD_TAlarm:=800);
	VRD05	:	obj_VRD_new 	:= (ID:=5, fFeedback:=TRUE, ReducedRange := FALSE,Local_VRD_TAlarm:=800);

	(* Temperature probes *)
	TPV01	:	obj_TPV := (ID:=1);
	TPV02	:	obj_TPV := (ID:=2, IN_WMIN:=50 , IN_WMAX:=800);
	TPV03	:	obj_TPV := (ID:=3, IN_WMIN:=50 , IN_WMAX:=800);
	TPV04	:	obj_TPV := (ID:=4);
	TPV05	:	obj_TPV := (ID:=5);
	TPV06	:	obj_TPV := (ID:=6);
	TPV07	:	obj_TPV := (ID:=7);
	TPV08	:	obj_TPV := (ID:=8);

	(* Zigbee temperature probes *)
	ZTHL09	:	obj_ZTHL := (ID:=1, Address:=17); (* ZTHL01 *)
	ZTHL10	:	obj_ZTHL := (ID:=2, Address:=12); (* ZTHL02 *)
	ZTHL11	:	obj_ZTHL := (ID:=3, Address:=13); (* ZTHL03 *)
	ZTHL12	:	obj_ZTHL := (ID:=4, Address:=14); (* ZTHL04 *)
	ZTHL13	:	obj_ZTHL := (ID:=5, Address:=15); (* ZTHL05 *)
	ZTHL14	:	obj_ZTHL := (ID:=6, Address:=16); (* ZTHL06 *)

	(** Communication **)
	(* ModBus *)
	MODB01	:	obj_MODBUS		:= (ID:=1, COM:=3, BAUDRATE:=BAUD_19200, RS485:=TRUE);
	MODB02	:	obj_MODBUS_TCP 	:= (ID:=1, IP:='192.168.100.4');

	(* M-Bus *)
	MBUS01	:	obj_MBUS		:= (ID:=1, COM:=2, BAUDRATE:=BAUD_2400);


	AggiornaLog: BOOL;


	(**** SIMULATION ONLY ****)
	(*...*)
END_VAR

(* Global variable list: LON/Module_1/InterfaceBlock_Module_1 *)
VAR_GLOBAL CONSTANT
(******************************************)
(* Automatic generated code, do not edit! *)
(******************************************)
	abSignature_Module_1 : ARRAY[0..15] OF BYTE := 16#1D,16#0B,16#57,16#52,16#5A,16#E8,16#6D,16#4B,16#89,16#27,16#1F,16#C7,16#5C,16#2F,16#78,16#C8;
	wConfigSize_Module_1 : WORD := 541;
	abInterface_Module_1 : ARRAY[0..135] OF DWORD :=
		16#D028C1F1, 16#210B060D, 16#6041B800, 16#06246830, 16#428B2E71, 16#64B95263, 16#FE000902, 16#2A050140, 
		16#00284095, 16#B2680DFC, 16#1C383063, 16#80015566, 16#CCD57140, 16#491D7775, 16#D5B152C7, 16#31D509A2, 
		16#D48882D5, 16#B8C2D6F1, 16#58664BDA, 16#129C49F3, 16#B7137DBE, 16#334D42A4, 16#13284D97, 16#A11A9D0A, 
		16#EC5BB754, 16#8A7D5A96, 16#DDB165D5, 16#251B7427, 16#B7794192, 16#0B526EDD, 16#6DDBBE1D, 16#92AEDBB2, 
		16#E596450B, 16#2D4C8065, 16#4A4D6BD7, 16#D9BA71CB, 16#B041776E, 16#15932F4C, 16#77EA5BF9, 16#EBD20D4B, 
		16#C9946573, 16#4D6B747E, 16#16C4CAB2, 16#065A4DD9, 16#3BA926E5, 16#7AE06C0A, 16#73B4BD85, 16#AD820478, 
		16#18B1AF54, 16#10554D2A, 16#B6D25295, 16#3E949D0A, 16#86651B94, 16#C01B6DE5, 16#CB56AAD1, 16#C09794C8, 
		16#0E452A4F, 16#D3AF3187, 16#634B0254, 16#A9229B03, 16#0DDCB665, 16#5C248436, 16#0BB7EE54, 16#46A65682, 
		16#F2A2594E, 16#46D29A10, 16#66FA28DC, 16#031AE0B4, 16#24A2A921, 16#E8CEC315, 16#12B88A94, 16#B14105CA, 
		16#58F608DD, 16#D3BE851A, 16#92402D6E, 16#216A74A8, 16#EBB6A8CC, 16#19D88A0D, 16#D2518944, 16#B31095DE, 
		16#EBCE48AD, 16#49C33B55, 16#A7422F59, 16#F39AD2D0, 16#D53C3E25, 16#7572E178, 16#8A066673, 16#40F93B2B, 
		16#0418102A, 16#FF000702, 16#10B08496, 16#A168016C, 16#64610830, 16#D908B0E2, 16#F005E684, 16#AED89C34, 
		16#9D9C1307, 16#83007FD6, 16#008D4EA0, 16#C64EA28E, 16#E0890497, 16#C9241020, 16#1510A0E0, 16#E0D5E009, 
		16#9C223CA9, 16#53862716, 16#B87E21AE, 16#D6E27AA5, 16#AE678CEB, 16#07B98E39, 16#EB9AE43A, 16#51AE6F93, 
		16#7A67B9EE, 16#9AEB01E6, 16#2E6CAE7F, 16#E7FAD0B9, 16#1BA1EBC5, 16#BA7E8CAE, 16#89E93A51, 16#AE23A8EB, 
		16#C3BABEA8, 16#EB8DEB3A, 16#C4AE2BB0, 16#BA33BBFE, 16#00EB51ED, 16#201C8A4F, 16#BA8C0990, 16#82543B63, 
		16#71C0A0CC, 16#70A0C080, 16#AF2EEC48, 16#2D7AAD52, 16#9E4CBCB4, 16#4BAEC73F, 16#0D8E1CEF, 16#00000050;
END_VAR

(* Global variable list: LON/Module_1/Runtime_Module_1 *)
VAR_GLOBAL
(******************************************)
(* Automatic generated code, do not edit! *)
(******************************************)
	mbxModule_1 : MBX_Full;
	InDataTelegram_Module_1 : ARRAY[0..255] OF BYTE;
	OutDataTelegram_Module_1 : ARRAY[0..511] OF BYTE;

	xInitRunning_Module_1 : BOOL := FALSE;
	unLastLen_mbxModule_1 : UINT;
END_VAR

(* Data type in LON/Enumerations *)
TYPE alarm_type_t :
(
	AL_HEADER := -13,
	AL_FOOTER := -12,
	AL_DEBUG := -11,
	AL_INFO := -10,
	AL_SYSTEM_INFO := -6,
	AL_VALUE_INVALID := -5,
	AL_CONSTANT := -4,
	AL_OFFLINE := -3,
	AL_UNKNOWN := -2,
	AL_NUL := -1,
	AL_NO_CONDITION := 0,
	AL_ALM_CONDITION := 1,
	AL_TOT_SVC_ALM_1 := 2,
	AL_TOT_SVC_ALM_2 := 3,
	AL_TOT_SVC_ALM_3 := 4,
	AL_LOW_LMT_CLR_1 := 5,
	AL_LOW_LMT_CLR_2 := 6,
	AL_HIGH_LMT_CLR_1 := 7,
	AL_HIGH_LMT_CLR_2 := 8,
	AL_LOW_LMT_ALM_1 := 9,
	AL_LOW_LMT_ALM_2 := 10,
	AL_HIGH_LMT_ALM_1 := 11,
	AL_HIGH_LMT_ALM_2 := 12,
	AL_FIR_ALM := 13,
	AL_FIR_PRE_ALM := 14,
	AL_FIR_TRBL := 15,
	AL_FIR_SUPV := 16,
	AL_FIR_TEST_ALM := 17,
	AL_FIR_TEST_PRE_ALM := 18,
	AL_FIR_ENVCOMP_MAX := 19,
	AL_FIR_MONITOR_COND := 20,
	AL_FIR_MAINT_ALERT := 21,
	AL_FATAL_ERROR := 30,
	AL_ERROR := 31,
	AL_WARNING := 32
);
END_TYPE

(* Data type in Logger *)
TYPE en_Logger_ErrLev :
(
	EL_Log			:=0,
	EL_Wrn			:=1,
	EL_Alarm		:=2,
	EL_AlarmStop	:=3
);
END_TYPE

(* Data type in Logger *)
TYPE en_Logger_Status :
(
	S_Logger_UNKNOWN := 0,
	S_Logger_IDLE,
	S_Logger_WAITCONN,
	S_Logger_WAITTX,
	S_Logger_WAITRESP,
	S_Logger_ERROR
);
END_TYPE

(* Data type *)
TYPE en_SYS_Objects :
(
	EO_SYS		:=0,  (* PLC *)
	EO_VPN		:=1,  (* VPN *)
	EO_DOOR		:=2,  (* Door & access control *)

	EO_CAL		:=10, (* Caldaia *)
	EO_CIR		:=11, (* Circolatore *)
	EO_CRON		:=12, (* Crono-termostato *)
	EO_VRD		:=13, (* Valvola miscelatore pannelli *)
	EO_CTL		:=14, (* Contalitri *)
	EO_CTB		:=15, (* Contabilizzatore *)
	EO_TPV		:=16, (* Temperature probes values *)
	EO_PPV		:=17, (* Pressure probes values *)
	EO_PBV		:=18, (* Over-Pressure Alarms *)
	EO_TBV		:=19, (* Over-Temperature Alarms *)
	EO_PMV		:=20, (* Under-Pressure Alarms *)
	EO_GRU		:=21, (* Gruppo termico *)
	EO_PDC		:=22, (* Pompa di calore *)
	EO_SOL		:=23, (* Pannello solare termico *)
	EO_ESOL		:=24, (* Pannello solare fotovoltaico *)
	EO_GAS		:=25, (* Contatore GAS *)
	EO_PORT		:=26, (* Misuratore di portata *)
	EO_FPV		:=27, (* Flow probes values *)
	EO_ANZ		:=28, (* Analizzatore di rete *)
	EO_SCA		:=29, (* Signal Control Alarms *)
	EO_LUX		:=30, (* Base Illumination point *)
	EO_LUXM		:=31, (* Metered Illumination point *)
	EO_PSG		:=32, (* Sensore di passaggio *)
	EO_HVAC		:=33, (* Heating, Ventilating and Air Conditioning *)
	EO_HYGRV	:=34, (* Relative Humidity sensors value *)
	EO_COOV		:=35, (* Carbon Dioxide CO2 sensors value *)
	EO_INV		:=36, (* Inverter *)
	EO_STR		:=37, (* Smart string box *)

	EO_CIRD		:=39, (* Double CIR *)
	EO_ACS		:=40, (* Hot domestic water *)
	EO_FRG		:=41, (* Frigo *)
	EO_THER		:=42, (* Thermostat *)
	EO_CIRM		:=43, (* Modbus CIR *)
	EO_CIRDM	:=44, (* Modbus double CIR *)

	EO_ZGW			:=200,  (* ZigBee - Gateway *)
	EO_ZRM			:=201,	(* ZigBee - Repeater *)
	EO_ZREL			:=202,	(* ZigBee - Actuator rele *)
	EO_ZTHL			:=203,	(* ZigBee - Temperature Sensor *)

	EO_ASGW			:=250,	(* ASi - Gateway *)
	EO_ASCBI		:=251,	(* ASi - Input Board, Ciabatta *)

	EO_LON			:=1000, (* Bus - LON *)
	EO_MODBUS		:=1001, (* Bus - MODBUS *)
	EO_MBUS			:=1002, (* Bus - M-BUS *)
	EO_MODBUS_TCP	:=1003, (* Bus - MODBUS TCP *)

	EO_GENERIC		:=9000, (* Generic dataset *)
	EO_EXPO			:=9001 (* EXPO dataset *)
);
END_TYPE

(* Data type *)
TYPE en_SYS_Status :
(
	S_UNKNOWN  := 0,
	S_STARTUP,
	S_INIT_RTC,
	S_INIT_VAR,
	S_AUTOTEST,
	S_RUNNING,
	S_SHUTDOWN,
	S_HALT
);
END_TYPE

(* Data type in LON/Enumerations *)
TYPE file_request_t :
(
	FR_NUL := -1,
	FR_OPEN_TO_SEND := 0,
	FR_OPEN_TO_RECEIVE := 1,
	FR_CLOSE_FILE := 2,
	FR_CLOSE_DELETE_FILE := 3,
	FR_DIRECTORY_LOOKUP := 4,
	FR_OPEN_TO_SEND_RA := 5,
	FR_OPEN_TO_RECEIVE_RA := 6
);
END_TYPE

(* Data type in LON/Enumerations *)
TYPE file_status_t :
(
	FS_NUL := -1,
	FS_XFER_OK := 0,
	FS_LOOKUP_OK := 1,
	FS_OPEN_FAIL := 2,
	FS_LOOKUP_ERR := 3,
	FS_XFER_UNDERWAY := 4,
	FS_IO_ERR := 5,
	FS_TIMEOUT_ERR := 6,
	FS_WINDOW_ERR := 7,
	FS_AUTH_ERR := 8,
	FS_ACCESS_UNAVAIL := 9,
	FS_SEEK_INVALID := 10,
	FS_SEEK_WAIT := 11
);
END_TYPE

(* Data type in LON/Enumerations *)
TYPE hvac_t :
(
	HVAC_NUL := -1,
	HVAC_AUTO := 0,
	HVAC_HEAT := 1,
	HVAC_MRNG_WRMUP := 2,
	HVAC_COOL := 3,
	HVAC_NIGHT_PURGE := 4,
	HVAC_PRE_COOL := 5,
	HVAC_OFF := 6,
	HVAC_TEST := 7,
	HVAC_EMERG_HEAT := 8,
	HVAC_FAN_ONLY := 9,
	HVAC_FREE_COOL := 10,
	HVAC_ICE := 11,
	HVAC_MAX_HEAT := 12,
	HVAC_ECONOMY := 13,
	HVAC_DEHUMID := 14,
	HVAC_CALIBRATE := 15,
	HVAC_EMERG_COOL := 16,
	HVAC_EMERG_STEAM := 17,
	HVAC_MAX_COOL := 18,
	HVAC_HVC_LOAD := 19,
	HVAC_NO_LOAD := 20
);
END_TYPE

(* Data type in LON/Enumerations *)
TYPE object_request_t :
(
	RQ_NUL := -1,
	RQ_NORMAL := 0,
	RQ_DISABLED := 1,
	RQ_UPDATE_STATUS := 2,
	RQ_SELF_TEST := 3,
	RQ_UPDATE_ALARM := 4,
	RQ_REPORT_MASK := 5,
	RQ_OVERRIDE := 6,
	RQ_ENABLE := 7,
	RQ_RMV_OVERRIDE := 8,
	RQ_CLEAR_STATUS := 9,
	RQ_CLEAR_ALARM := 10,
	RQ_ALARM_NOTIFY_ENABLED := 11,
	RQ_ALARM_NOTIFY_DISABLED := 12,
	RQ_MANUAL_CTRL := 13,
	RQ_REMOTE_CTRL := 14,
	RQ_PROGRAM := 15,
	RQ_CLEAR_RESET := 16,
	RQ_RESET := 17,
	RQ_CLEAR_LOG := 18,
	RQ_LOAD_PROGRAM := 19,
	RQ_RUN_PROGRAM := 20,
	RQ_HALT_PROGRAM := 21,
	RQ_RESTART_PROGRAM := 22,
	RQ_UNLOAD_PROGRAM := 23,
	RQ_STEP_PROGRAM := 24
);
END_TYPE

(* Data type in LON/Enumerations *)
TYPE priority_level_t :
(
	PR_NUL := -1,
	PR_LEVEL_0 := 0,
	PR_LEVEL_1 := 1,
	PR_LEVEL_2 := 2,
	PR_LEVEL_3 := 3,
	PR_1 := 4,
	PR_2 := 5,
	PR_3 := 6,
	PR_4 := 7,
	PR_6 := 8,
	PR_8 := 9,
	PR_10 := 10,
	PR_16 := 11
);
END_TYPE

(* Data type in Plant_Objects *)
TYPE typ_Clima : (* CURVA CLIMATICA *)
STRUCT
	InitOK:		BOOL;
	Points: 	ARRAY [0..10] OF POINT;
END_STRUCT
END_TYPE

(* Data type in Plant_Objects *)
TYPE typ_Cron_Calendar :
STRUCT
	Profile		: ARRAY[0..384] OF BYTE;
END_STRUCT
END_TYPE

(* Data type in Plant_Objects *)
TYPE typ_Cron_Jolly :
STRUCT
	Start		: DT;
	End			: DT;
	Temp		: WORD;
	Flags		: WORD; (* B0:Enabled B1..B15:Unused *)
END_STRUCT
END_TYPE

(* Data type in Plant_Objects *)
TYPE typ_Cron_Profile :
STRUCT
	Flags		: WORD;
	Setpoint	: ARRAY [0..95] OF WORD;
END_STRUCT
END_TYPE

(* Data type in Plant_Objects *)
TYPE typ_Frigo :
STRUCT
	Status	:	BOOL;		(* 0=OFF, 1=ON	*)
	Mode	:	BOOL;		(* 0=COLD, 1=HOT	*)

END_STRUCT
END_TYPE

(* Data type in Logger *)
TYPE typ_Logger :
STRUCT
	Status		: en_Logger_Status;

	SendReq		: BOOL;
	SendIdx		: DWORD;
	SendData	: ARRAY [0..MAX_SEND_TCP_CLIENT] OF BYTE;
	SendLen		: DINT;

	TData		: ARRAY [0..MAX_SEND_TCP_CLIENT] OF BYTE;
	TLen		: DINT;

	LastIdxPos	: DWORD;

	(* Temporary variables used by objects *)
	s1			: STRING(256);
	i1			: WORD;

END_STRUCT
END_TYPE

(* Data type in Plant_Objects *)
TYPE typ_MODBUS_CIR :
STRUCT
	PumpStatus		:	WORD;
	PumpFault		:	BOOL;
	PumpBoardTemp	:	INT;	(* Electonic board temperature  [°C] *)
	PumpVoltage		:	WORD;	(* Input voltage rms [V] *)
	PumpCurrent		:	WORD;	(* Output current [E-3 A]	*)
	PumpRPM			:	WORD;	(* Round per minute [rpm] *)
	PumpPower		:	WORD;	(* Power [W] *)
	PumpOpTime		:	DWORD;	(* Pump operating time [h] *)
	PumpHead		:	WORD;	(* [E-1 m] *)
	PumpFlow		:	WORD;	(* Extimated flow [E-1 m3/h] *)
	PumpLiqTemp		:	WORD;	(* Liquid temperature [°C] *)
	PumpAlarm		:	ARRAY [0..14] OF WORD;

END_STRUCT
END_TYPE

(* Data type in Plant_Objects *)
TYPE typ_MODBUS_VAR : (* Gestione parametri MODBUS *)
STRUCT
	SlaveAddress	: BYTE;
	FunCode			: BYTE;
	FunAddress		: WORD;
	Refresh_Time	: BYTE; (* 0:No refresh x:Refresh in seconds *)
	Refresh_Cnt		: BYTE; (* INTERNAL *)
	Variable		: POINTER TO WORD;
	Variable_Size	: BYTE;
	Variable_Mirror : WORD; (* INTERNAL [Force refresh on read variables when <>0] *)
END_STRUCT
END_TYPE

(* Data type *)
TYPE typ_SYS :
STRUCT
	Status			: en_SYS_Status;
	Warning			: BOOL;
	Alarm			: BOOL;
	AlarmStop		: BOOL;

	Time_LogString	: STRING;
	Time_Year		: WORD;
	Time_Month		: BYTE;
	Time_Day		: BYTE;
	Time_Hour		: BYTE;
	Time_Minute		: BYTE;

	Time_CT_DT		: DT;
	Time_CT_Day		: WORD;
	Time_CT_Quarter	: BYTE;

	LastLogs_Idx	: BYTE;
	LastLogs_Dat	: ARRAY[0..5] OF STRING;
	LastLogs_Msg	: ARRAY[0..5] OF STRING;

END_STRUCT
END_TYPE

(* Data type in Plant_Objects *)
TYPE typ_VisuStrutturaMbus :
STRUCT

	sdNodoPresente: STRING(16);
	sdEnergia: STRING(16);
	sdPotenza: STRING(16);
	sdVolume: STRING(16);
	sdFlow: STRING(16);
	sdTempIngresso: STRING(8);
	sdTempaUscita: STRING(8);
	sdTempDelta: STRING(8);

END_STRUCT
END_TYPE

(* Data type in LON/NetworkVariables *)
TYPE typSnvtAlarm : 
STRUCT
	abLocation : ARRAY[0..5] OF BYTE;
	wObjectId : WORD;
	bAlarmType : BYTE (* enum type alarm_type_t *);
	bPriorityLevel : BYTE (* enum type priority_level_t *);
	wIndexToSnvt : WORD;
	abValue : ARRAY[0..3] OF BYTE;
	wYear : WORD;
	bMonth : BYTE;
	bDay : BYTE;
	bHour : BYTE;
	bMinute : BYTE;
	bSecond : BYTE;
	wMillisecond : WORD;
	abAlarmLimit : ARRAY[0..3] OF BYTE;
	bStatusInformation : BYTE; (* bit allocation of bStatusInformation:
	bit 0: NVI update counter LSB
	bit 1: NVI update counter
	bit 2: NVI update counter
	bit 3: NVI update counter MSB
	bit 4: timeout for NVI occurs (MaxRcvTime expired)
	bit 5: reserved
	bit 6: reserved
	bit 7: force NVO update *)
	bInternalUseOnly : BYTE; (* Do not use this byte in your application! *)
END_STRUCT
END_TYPE

(* Data type in LON/NetworkVariables *)
TYPE typSnvtFilePos : 
STRUCT
	diRwPtr : DINT;
	wRwLength : WORD;
	bStatusInformation : BYTE; (* bit allocation of bStatusInformation:
	bit 0: NVI update counter LSB
	bit 1: NVI update counter
	bit 2: NVI update counter
	bit 3: NVI update counter MSB
	bit 4: timeout for NVI occurs (MaxRcvTime expired)
	bit 5: reserved
	bit 6: reserved
	bit 7: force NVO update *)
	bInternalUseOnly : BYTE; (* Do not use this byte in your application! *)
END_STRUCT
END_TYPE

(* Data type in LON/NetworkVariables *)
TYPE typSnvtFileReq : 
STRUCT
	bRequest : BYTE (* enum type file_request_t *);
	wIndex : WORD;
	wReceiveTimeout : WORD;
	abDestAddress : ARRAY[0..4] OF BYTE (* union declaration *);
	bAuthOn : BYTE;
	bPrioOn : BYTE;
	bStatusInformation : BYTE; (* bit allocation of bStatusInformation:
	bit 0: NVI update counter LSB
	bit 1: NVI update counter
	bit 2: NVI update counter
	bit 3: NVI update counter MSB
	bit 4: timeout for NVI occurs (MaxRcvTime expired)
	bit 5: reserved
	bit 6: reserved
	bit 7: force NVO update *)
	bInternalUseOnly : BYTE; (* Do not use this byte in your application! *)
END_STRUCT
END_TYPE

(* Data type in LON/NetworkVariables *)
TYPE typSnvtFileStatus : 
STRUCT
	bStatus : BYTE (* enum type file_status_t *);
	wNumberOfFiles : WORD;
	wSelectedFile : WORD;
	abAdr : ARRAY[0..21] OF BYTE (* union declaration *);
	bStatusInformation : BYTE; (* bit allocation of bStatusInformation:
	bit 0: NVI update counter LSB
	bit 1: NVI update counter
	bit 2: NVI update counter
	bit 3: NVI update counter MSB
	bit 4: timeout for NVI occurs (MaxRcvTime expired)
	bit 5: reserved
	bit 6: reserved
	bit 7: force NVO update *)
	bInternalUseOnly : BYTE; (* Do not use this byte in your application! *)
END_STRUCT
END_TYPE

(* Data type in LON/NetworkVariables *)
TYPE typSnvtHvacMode : 
STRUCT
	bSnvtHvacMode : BYTE (* enum type hvac_t *);
	bStatusInformation : BYTE; (* bit allocation of bStatusInformation:
	bit 0: NVI update counter LSB
	bit 1: NVI update counter
	bit 2: NVI update counter
	bit 3: NVI update counter MSB
	bit 4: timeout for NVI occurs (MaxRcvTime expired)
	bit 5: reserved
	bit 6: reserved
	bit 7: force NVO update *)
	bInternalUseOnly : BYTE; (* Do not use this byte in your application! *)
END_STRUCT
END_TYPE

(* Data type in LON/NetworkVariables *)
TYPE typSnvtObjRequest : 
STRUCT
	wObjectId : WORD;
	bObjectRequest : BYTE (* enum type object_request_t *);
	bStatusInformation : BYTE; (* bit allocation of bStatusInformation:
	bit 0: NVI update counter LSB
	bit 1: NVI update counter
	bit 2: NVI update counter
	bit 3: NVI update counter MSB
	bit 4: timeout for NVI occurs (MaxRcvTime expired)
	bit 5: reserved
	bit 6: reserved
	bit 7: force NVO update *)
	bInternalUseOnly : BYTE; (* Do not use this byte in your application! *)
END_STRUCT
END_TYPE

(* Data type in LON/NetworkVariables *)
TYPE typSnvtObjStatus : 
STRUCT
	wObjectId : WORD;
	bBitfieldByteOffset2 : BYTE (* bit field *);
	bBitfieldByteOffset3 : BYTE (* bit field *);
	bBitfieldByteOffset4 : BYTE (* bit field *);
	bBitfieldByteOffset5 : BYTE (* bit field *);
	bStatusInformation : BYTE; (* bit allocation of bStatusInformation:
	bit 0: NVI update counter LSB
	bit 1: NVI update counter
	bit 2: NVI update counter
	bit 3: NVI update counter MSB
	bit 4: timeout for NVI occurs (MaxRcvTime expired)
	bit 5: reserved
	bit 6: reserved
	bit 7: force NVO update *)
	bInternalUseOnly : BYTE; (* Do not use this byte in your application! *)
END_STRUCT
END_TYPE

(* Data type in LON/NetworkVariables *)
TYPE typSnvtState : 
STRUCT
	bBitfieldByteOffset0 : BYTE (* bit field *);
	bBitfieldByteOffset1 : BYTE (* bit field *);
	bStatusInformation : BYTE; (* bit allocation of bStatusInformation:
	bit 0: NVI update counter LSB
	bit 1: NVI update counter
	bit 2: NVI update counter
	bit 3: NVI update counter MSB
	bit 4: timeout for NVI occurs (MaxRcvTime expired)
	bit 5: reserved
	bit 6: reserved
	bit 7: force NVO update *)
	bInternalUseOnly : BYTE; (* Do not use this byte in your application! *)
END_STRUCT
END_TYPE

(* Data type in LON/NetworkVariables *)
TYPE typSnvtSwitch : 
STRUCT
	bValue : BYTE;
	siState : SINT;
	bStatusInformation : BYTE; (* bit allocation of bStatusInformation:
	bit 0: NVI update counter LSB
	bit 1: NVI update counter
	bit 2: NVI update counter
	bit 3: NVI update counter MSB
	bit 4: timeout for NVI occurs (MaxRcvTime expired)
	bit 5: reserved
	bit 6: reserved
	bit 7: force NVO update *)
	bInternalUseOnly : BYTE; (* Do not use this byte in your application! *)
END_STRUCT
END_TYPE

(* Data type in LON/NetworkVariables *)
TYPE typSnvtTempP : 
STRUCT
	iSnvtTempP : INT;
	bStatusInformation : BYTE; (* bit allocation of bStatusInformation:
	bit 0: NVI update counter LSB
	bit 1: NVI update counter
	bit 2: NVI update counter
	bit 3: NVI update counter MSB
	bit 4: timeout for NVI occurs (MaxRcvTime expired)
	bit 5: reserved
	bit 6: reserved
	bit 7: force NVO update *)
	bInternalUseOnly : BYTE; (* Do not use this byte in your application! *)
END_STRUCT
END_TYPE

(* Data type in LON/NetworkVariables *)
TYPE typSnvtTimeStamp : 
STRUCT
	iYear : INT;
	bMonth : BYTE;
	bDay : BYTE;
	bHour : BYTE;
	bMinute : BYTE;
	bSecond : BYTE;
	bStatusInformation : BYTE; (* bit allocation of bStatusInformation:
	bit 0: NVI update counter LSB
	bit 1: NVI update counter
	bit 2: NVI update counter
	bit 3: NVI update counter MSB
	bit 4: timeout for NVI occurs (MaxRcvTime expired)
	bit 5: reserved
	bit 6: reserved
	bit 7: force NVO update *)
	bInternalUseOnly : BYTE; (* Do not use this byte in your application! *)
END_STRUCT
END_TYPE

(* POU PLC_PRG, ST *)
PROGRAM PLC_PRG
VAR
	Timer1: TON; (* Fast controls tick *)
	Timer2: TON; (* Plant control tick *)
	Timer3: TON; (* Logger timer *)

	T_CIR01		:	INT;
	T_CIR02		:	INT;
	T_CIR03		:	INT;
	T_CIRD01	:	INT;
	T_CIRD02	:	INT;

	T_Valve01	:	INT;
	T_Valve02	:	INT;
	T_Valve03	:	INT;
	T_Valve04	:	INT;
	T_Valve05	:	INT;

	SecCircuitLogic	:	BOOL;	(* Secondary circuit request: LOGICAL ON/OFF *)
	SecCircuitReal	:	BOOL;	(* Secondart circuit request: REAL ON/OFF	 *)

	i	:	INT;


	StartCAL_Antigelo: RS;
	fAntigelo		:FLT_TAP;  (* Sgnalazione LOG Antigelo  *)


END_VAR
(******************************************************************************
 ****                           MAIN TASK CODE                             ****
 ******************************************************************************

	Network setup:
		IP  = 192.168.100.2 | MSK = 255.255.255.0
		GW	= 192.168.100.1 | DNS = 192.168.100.1
		SNTP = 193.204.114.232 (3600s) ==> 192.168.100.3

*)

(*==============================*)
(*===== Main status machine ====*)
(*==============================*)
Main_Stm();

(*==============================*)
(*== Running cycle operations ==*)
(*==============================*)
IF SYS.Status>S_INIT_VAR THEN
	(* Execute cycle processes *)
	(* Update LON output variables (needs to be here to obtain only one refresh) *)
	GRU01.Heartbeat( CLIM:=GRU01_Clima );
	(* Execute LON process *)
	Module_1_PRG();

	(* Count water pulses *)
	CTL01(CTL_ST:=CTL01_ST, COUNT:=Ctl01_Counter);
	CTL02(CTL_ST:=CTL02_ST, COUNT:=Ctl02_Counter);

	(* ModBus *)
	MODB01();

		(*	CIR01 (Pump_AL:=NOT CIR01_AL , Pump_ST:=CIR01_ST , Pump_AUTO:=CIR01_AUTO, CIR_EN=>CIR01_EN );
			CIR02 (Pump_AL:=NOT CIR02_AL , Pump_ST:=CIR02_ST , Pump_AUTO:=CIR02_AUTO, CIR_EN=>CIR02_EN ); *)



	CIR03(ModBus:=MODB01, Pump_AL:=NOT CIR03_AL, Pump_AUTO:=NOT CIR03_AUTO);

	CIRD01(ModBus:=MODB01, PumpA_AL:=NOT CIRD01_A_AL, PumpB_AL:=NOT CIRD01_B_AL, PumpA_AUTO:=NOT CIRD01_A_AUTO, PumpB_AUTO:=NOT CIRD01_B_AUTO);
	CIRD02(ModBus:=MODB01, PumpA_AL:=NOT CIRD02_A_AL, PumpB_AL:=NOT CIRD02_B_AL, PumpA_AUTO:=NOT CIRD02_A_AUTO, PumpB_AUTO:=NOT CIRD02_B_AUTO);

NodoDaInterrogare:=LIMIT(1,NodoDaInterrogare,6);
IF NodoDaInterrogare>5 THEN NodoDaInterrogare:=1;END_IF;


	(* TCP ModBus *)
	MODB02();

	ZTHL09(MODBUS:=MODB02);
	ZTHL10(MODBUS:=MODB02);
	ZTHL11(MODBUS:=MODB02);
	ZTHL12(MODBUS:=MODB02);
	ZTHL13(MODBUS:=MODB02);
	ZTHL14(MODBUS:=MODB02);

	(* M-Bus *)
	MBUS01();

	CTB01(MBUS:=MBUS01);
	CTB02(MBUS:=MBUS01);

END_IF

(*==============================*)
(*== System cycle operations ===*)
(*==============================*)
(* Execute TCP processes *)
Logger_Proc();
Remote_Proc();
(* Update user led *)
USRLED_Update();
(* Execute Cron Editor commands *)
CronEd();

(* Environment temperature *)
IF NOT TPV01.ERR THEN T_AMB := S01;
ELSE T_AMB := Plant_DefaultTAmb;
END_IF


(**** SIMULATION ONLY ****)
(*...*)
END_PROGRAM
ACTION Main_Stm:
CASE Sys.Status OF

	S_STARTUP:
		Sys.Status:=S_INIT_RTC;

	S_INIT_RTC:
		(* Check RTC and update from network *)
		RTC_Update();
		(* Check time *)
		IF Sys.Time_Year>2000 THEN
			Sys.Status:=S_INIT_VAR;
		END_IF

	S_INIT_VAR:
		LogEv(EL_Wrn,EO_SYS,0,1,CONCAT('System_startup_v',WORD_TO_STRING(Plant_SW_VER)));
		Sys.Status:=S_RUNNING;

	S_RUNNING:
		Timer1(IN:=NOT Timer1.Q,PT:=T#50ms);
		IF Timer1.Q THEN
			(* Update meters *)

			(* Update system checks *)
			SYS_Proc();
		END_IF

		Timer2(IN:=NOT Timer2.Q,PT:=T#500ms);
		IF Timer2.Q THEN
			(* Read current date/time *)
			RTC_Update();


			(* Probes *)
			TPV01(IN:=S01);
			TPV02(IN:=S02);
			TPV03(IN:=S03);
			TPV04(IN:=S04);
			TPV05(IN:=S05);
			TPV06(IN:=S06);
			TPV07(IN:=S07);
			TPV08(IN:=S08);








(*		i := 2 - (BOOL_TO_INT(ZTHL13.ERR)+BOOL_TO_INT(ZTHL14.ERR));

			IF i=0 THEN T_CIRD02 := Plant_DefaultTAmb;
			ELSE T_CIRD02 := (ZTHL13.OUT_TEMP + ZTHL14.OUT_TEMP)/i;
			END_IF
*)
			T_Valve01 := SEL(TPV04.ERR,TPV04.AVG,Plant_VRD_TDefault);
			T_Valve02 := SEL(TPV05.ERR,TPV05.AVG,Plant_VRD_TDefault);

			T_Valve03 := SEL(TPV06.ERR,TPV06.AVG,Plant_VRD_TDefault);

			T_Valve04 := SEL(TPV07.ERR,TPV07.AVG,Plant_VRD_TDefault);

			T_Valve05 := SEL(TPV08.ERR,TPV08.AVG,Plant_VRD_TDefault);



		(* Gestione Ciclo antigelo : in questo impianto il ciclo antigelo è gestito coi crono ambiente *)

			StartCAL_Antigelo(	SET:=(SogliaMinStartAntigelo>TPV03.AVG),
								RESET1:= (TPV03.AVG>SogliaMinStopAntigelo) OR NOT BitAbilitaAntigelo
							);

			fAntigelo(IN:=StartCAL_Antigelo.Q1);
			IF fAntigelo.EVH THEN
				LogEv(EL_Log,EO_SYS,0,11,'Ciclo_Antigelo_Attivato');
			END_IF
			IF fAntigelo.EVL THEN
				LogEv(EL_Log,EO_SYS,0,12,'Ciclo_Antigelo_Disattivato');
			END_IF



			(* Thermostats *)
			T_CIR01 := ZTHL11.OUT_TEMP;  	(* Auditorium  *)
			THER01(Temperature:=T_CIR01);
			CIR01.OnOff:= SEL(ZTHL11.ERR,THER01.Run,THER01.RunCrono) OR StartCAL_Antigelo.Q1;

			T_CIR02 := ZTHL09.OUT_TEMP;  	(* Aula Disegnao *)
			THER02(Temperature:=T_CIR02);(*, AntifreezeForce=>CIR02.CIR_RUN_REQ);*)
			CIR02.OnOff:= SEL(ZTHL09.ERR,THER02.Run,THER02.RunCrono) OR StartCAL_Antigelo.Q1;

			(* Limito la lettura della sonda temperatura per evitare dissevizi *)
			T_CIR03 := ZTHL12.OUT_TEMP;		(* Piano 1 Liceo *)
			T_CIR03 := MIN (T_CIR03,ZTHL14.OUT_TEMP);
			THER03(Temperature:=T_CIR03, Run=>);(*, AntifreezeForce=>CIR03.CIR_RUN_REQ);*)
			CIR03.OnOff:= SEL(ZTHL12.ERR AND ZTHL14.ERR ,THER03.Run,THER03.RunCrono) OR StartCAL_Antigelo.Q1;

			T_CIRD01 := ZTHL10.OUT_TEMP;  	(* Aule IPD  *)
			THER04(Temperature:=T_CIRD01);(*, AntifreezeForce=>CIRD01.CIR_RUN_REQ);*)
			CIRD01.OnOff:=SEL(ZTHL10.ERR,THER04.Run,THER04.RunCrono) OR StartCAL_Antigelo.Q1;

			T_CIRD02 := ZTHL13.OUT_TEMP;  	(* Mansarde Liceo *)
			THER05(Temperature:=T_CIRD02, Run=>);(*, AntifreezeForce=>CIRD02.CIR_RUN_REQ);*)
			CIRD02.OnOff:=SEL(ZTHL13.ERR,THER05.Run,THER05.RunCrono) OR StartCAL_Antigelo.Q1;

			THER250();

			(* CIR *)
			CIR01(Pump_AL:=NOT CIR01_AL, Pump_ST:=CIR01_ST, Pump_AUTO:=NOT CIR01_AUTO, CIR_EN=>CIR01_EN);
			CIR02(Pump_AL:=NOT CIR02_AL, Pump_ST:=CIR02_ST, Pump_AUTO:=NOT CIR02_AUTO, CIR_EN=>CIR02_EN);

			(* Valves *)
			VRD01(RUN:=CIRD02.Run,OffsetBoost:=THER250.SetPoint, CLIM:=VRD01_Clima, TEMP:=T_Valve01, STATUS:=VRD01_ST, OUT_CL=>VRD01_CL, OUT_OP=>VRD01_OP);
			VRD02(RUN:=CIR03.Run,OffsetBoost:=THER250.SetPoint, CLIM:=VRD02_Clima, TEMP:=T_Valve02, STATUS:=VRD02_ST, OUT_CL=>VRD02_CL, OUT_OP=>VRD02_OP);
			VRD03(RUN:=CIRD01.Run,OffsetBoost:=THER250.SetPoint, CLIM:=VRD03_Clima, TEMP:=T_Valve03, STATUS:=VRD03_ST, OUT_CL=>VRD03_CL, OUT_OP=>VRD03_OP);
			VRD04(RUN:=CIR02.Run,OffsetBoost:=THER250.SetPoint, CLIM:=VRD04_Clima, TEMP:=T_Valve04, STATUS:=VRD04_ST, OUT=>VRD04_CTRL);
			VRD05(RUN:=CIR01.Run,OffsetBoost:=THER250.SetPoint, CLIM:=VRD05_Clima, TEMP:=T_Valve05, STATUS:=VRD05_ST, OUT=>VRD05_CTRL);



			(* Secondary circuit heat request *)
			SecCircuitLogic := CIR01.Ctrl_Run OR CIR02.Ctrl_Run OR CIR03.Ctrl_Run OR CIRD01.Ctrl_Run OR CIRD02.Ctrl_Run;
			SecCircuitReal	:= CIR01.Run OR CIR02.Run OR CIR03.Run OR CIRD01.Run OR CIRD02.Run;

			GRU01.Run := SEL(SecCircuitLogic,FALSE,TRUE) AND SYS.AlarmStop=FALSE;

			(* Scrivo il setpoint in funzione della curva cliamatica più alta *)



			GRU01.SetPointManuale:=GRU01.Curve_Temp - OffsetSetPointManuale + THER250.SetPoint;
			GRU01.SetPointManuale:=MAX(GRU01.SetPointManuale,SEL(VRD01.RUN,0,VRD01.Ctrl_SetPoint));
			GRU01.SetPointManuale:=MAX(GRU01.SetPointManuale,SEL(VRD02.RUN,0,VRD02.Ctrl_SetPoint));
			GRU01.SetPointManuale:=MAX(GRU01.SetPointManuale,SEL(VRD03.RUN,0,VRD03.Ctrl_SetPoint));
			GRU01.SetPointManuale:=MAX(GRU01.SetPointManuale,SEL(VRD04.RUN,0,VRD04.Ctrl_SetPoint));
			GRU01.SetPointManuale:=MAX(GRU01.SetPointManuale,SEL(VRD05.RUN,0,VRD05.Ctrl_SetPoint));


			GRU01(CLIM:=GRU01_Clima,AbilitaSetPointManuale:=TRUE);



			(* Check plant status *)

			Lamp( Allarme:=	GRU01.Status_Log=2 OR
  						  	CIR01.Status_Log=2 OR
  						  	CIR02.Status_Log=2 OR
  						  	CIR03.Status_Log=2 OR
 						  	CIRD01.Status_Log=2 OR
						  	CIRD02.Status_Log=2 OR
							TPV01.Status_Log=2 OR
							TPV02.Status_Log=2 OR
							TPV03.Status_Log=2 OR
							TPV04.Status_Log=2 OR
							TPV05.Status_Log=2 OR
							TPV06.Status_Log=2 OR
							TPV07.Status_Log=2 OR
							TPV08.Status_Log=2 OR
							THER01.Status_Log=2 OR
							THER02.Status_Log=2 OR
							THER03.Status_Log=2 OR
							THER04.Status_Log=2 OR
							THER05.Status_Log=2 OR
							THER250.Status_Log=2 OR
							VRD01.Status_Log=2 OR
							VRD02.Status_Log=2 OR
							VRD03.Status_Log=2 OR
							VRD04.Status_Log=2 OR
							VRD05.Status_Log=2 OR
							CTL01.Status_Log=2 OR
							CTL02.Status_Log=2 OR
							CTB01.Status_Log=2 OR
							CTB02.Status_Log=2 OR
							MODB01.Status_Log=2 OR
							MODB02.Status_Log=2 OR
							MBUS01.Status_Log=2 OR
							ZTHL09.Status_Log=2 OR
							ZTHL10.Status_Log=2 OR
							ZTHL11.Status_Log=2 OR
							ZTHL12.Status_Log=2 OR
							ZTHL13.Status_Log=2 OR
							ZTHL14.Status_Log=2 ,
							Warning:=GRU01.Status_Log=1 OR
  						  	CIR01.Status_Log=1 OR
  						  	CIR02.Status_Log=1 OR
  						  	CIR03.Status_Log=1 OR
 						  	CIRD01.Status_Log=1 OR
						  	CIRD02.Status_Log=1 OR
							TPV01.Status_Log=1 OR
							TPV02.Status_Log=1 OR
							TPV03.Status_Log=1 OR
							TPV04.Status_Log=1 OR
							TPV05.Status_Log=1 OR
							TPV06.Status_Log=1 OR
							TPV07.Status_Log=1 OR
							TPV08.Status_Log=1 OR
							THER01.Status_Log=1 OR
							THER02.Status_Log=1 OR
							THER03.Status_Log=1 OR
							THER04.Status_Log=1 OR
							THER05.Status_Log=1 OR
							THER250.Status_Log=1 OR
							VRD01.Status_Log=1 OR
							VRD02.Status_Log=1 OR
							VRD03.Status_Log=1 OR
							VRD04.Status_Log=1 OR
							VRD05.Status_Log=1 OR
							CTL01.Status_Log=1 OR
							CTL02.Status_Log=1 OR
							CTB01.Status_Log=1 OR
							CTB02.Status_Log=1 OR
							MODB01.Status_Log=1 OR
							MODB02.Status_Log=1 OR
							MBUS01.Status_Log=1 OR
							ZTHL09.Status_Log=1 OR
							ZTHL10.Status_Log=1 OR
							ZTHL11.Status_Log=1 OR
							ZTHL12.Status_Log=1 OR
							ZTHL13.Status_Log=1 OR
							ZTHL14.Status_Log=1	,
							AllarmeLampada=>LAMP_AL
							);






















			(* Test toggle *)
			(*IF TEST1 THEN TEST1:=FALSE; ELSE TEST1:=TRUE; END_IF*)
		END_IF

		Timer3(IN:=NOT Timer3.Q,PT:=T#5m);
		IF Timer3.Q OR AggiornaLog THEN
			(* Trig logger *)
			LogTrig();
			(* Execute temporary CSV logger *)
			(*CSV_Log();*)
		END_IF

	S_SHUTDOWN:
		(* Stop sistema *)
		Sys.Status:=S_STARTUP;

	S_HALT:
		(* Aspetta uscita manuale *)
		Sys.Status:=S_STARTUP;

ELSE
	Sys.Status:=S_STARTUP;
END_CASE;
END_ACTION

(* POU Utils Functions/FLT_TAP, ST *)
FUNCTION_BLOCK FLT_TAP
VAR_INPUT
	IN		: BOOL;
	TAP		: BYTE:=4;
	INITEV	: BOOL:=TRUE;
END_VAR
VAR_OUTPUT
	OUT		: BOOL;
	EVH		: BOOL;
	EVL		: BOOL;
END_VAR
VAR
	init	: BOOL:=FALSE;
	cnt		: BYTE;
END_VAR
EVH:=FALSE;
EVL:=FALSE;

IF NOT init THEN
	init := TRUE;
	IF INITEV THEN
		OUT  := NOT IN;
		cnt  := TAP;
	ELSE
		OUT  := IN;
	END_IF
END_IF

IF OUT<>IN THEN
	cnt:=cnt+1;
	IF cnt>TAP THEN
		OUT:=IN;
		cnt:=0;
		IF OUT THEN EVH:=TRUE; ELSE EVL:=TRUE; END_IF
	END_IF
ELSE
	cnt:=0;
END_IF
END_FUNCTION_BLOCK

(* POU LON/Module_1/Module_1_PRG, FBD *)
PROGRAM Module_1_PRG
VAR
	(* Automatic added code, do not change! *)
	LonMaster : Module_1_LonMaster;
	SFPTnodeObject : Module_1_SFPTnodeObject;
	Virtualfunctionalblock : Module_1_Virtualfunctionalblock;

	InData_LON AT %IB4 : ARRAY[0..23] OF BYTE;
	OutData_LON AT %QB0 : ARRAY[0..23] OF BYTE;
	(***** End of automatic added code. *****)

	(* Add your code here. *)
	LonState: BOOL;
	LonReset: BOOL;

END_VAR
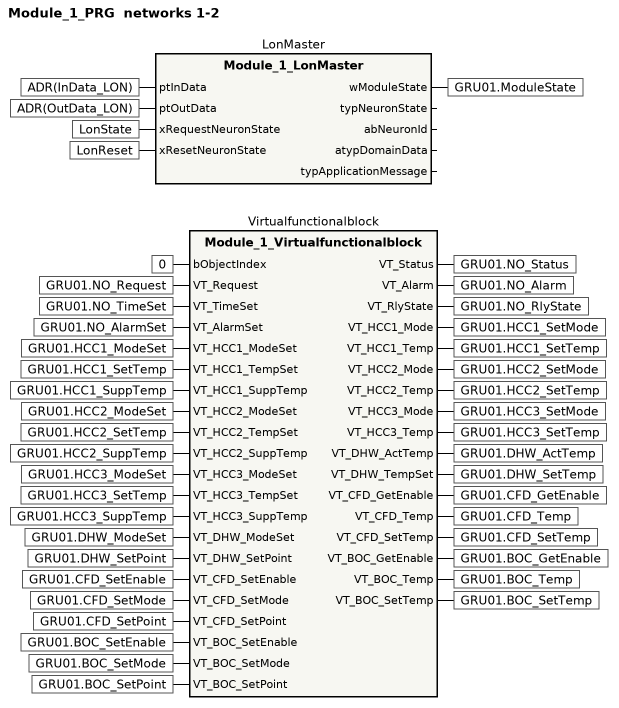
_FBD_ (* Function Block Diagram *)
NETWORK 1 (* Added by code generator *)
	LonMaster:Module_1_LonMaster(ptInData: ADR(InData_LON), ptOutData: ADR(OutData_LON), xRequestNeuronState: LonState, xResetNeuronState: LonReset) => GRU01.ModuleState
NETWORK 2
	Virtualfunctionalblock:Module_1_Virtualfunctionalblock(bObjectIndex: 0, VT_Request: GRU01.NO_Request, VT_TimeSet: GRU01.NO_TimeSet, VT_AlarmSet: GRU01.NO_AlarmSet, VT_HCC1_ModeSet: GRU01.HCC1_ModeSet, VT_HCC1_TempSet: GRU01.HCC1_SetTemp, VT_HCC1_SuppTemp: GRU01.HCC1_SuppTemp, VT_HCC2_ModeSet: GRU01.HCC2_ModeSet, VT_HCC2_TempSet: GRU01.HCC2_SetTemp, VT_HCC2_SuppTemp: GRU01.HCC2_SuppTemp, VT_HCC3_ModeSet: GRU01.HCC3_ModeSet, VT_HCC3_TempSet: GRU01.HCC3_SetTemp, VT_HCC3_SuppTemp: GRU01.HCC3_SuppTemp, VT_DHW_ModeSet: GRU01.DHW_ModeSet, VT_DHW_SetPoint: GRU01.DHW_SetPoint, VT_CFD_SetEnable: GRU01.CFD_SetEnable, VT_CFD_SetMode: GRU01.CFD_SetMode, VT_CFD_SetPoint: GRU01.CFD_SetPoint, VT_BOC_SetEnable: GRU01.BOC_SetEnable, VT_BOC_SetMode: GRU01.BOC_SetMode, VT_BOC_SetPoint: GRU01.BOC_SetPoint, VT_Alarm => GRU01.NO_Alarm, VT_RlyState => GRU01.NO_RlyState, VT_HCC1_Mode => GRU01.HCC1_SetMode, VT_HCC1_Temp => GRU01.HCC1_SetTemp, VT_HCC2_Mode => GRU01.HCC2_SetMode, VT_HCC2_Temp => GRU01.HCC2_SetTemp, VT_HCC3_Mode => GRU01.HCC3_SetMode, VT_HCC3_Temp => GRU01.HCC3_SetTemp, VT_DHW_ActTemp => GRU01.DHW_ActTemp, VT_DHW_TempSet => GRU01.DHW_SetTemp, VT_CFD_GetEnable => GRU01.CFD_GetEnable, VT_CFD_Temp => GRU01.CFD_Temp, VT_CFD_SetTemp => GRU01.CFD_SetTemp, VT_BOC_GetEnable => GRU01.BOC_GetEnable, VT_BOC_Temp => GRU01.BOC_Temp, VT_BOC_SetTemp => GRU01.BOC_SetTemp) => GRU01.NO_Status
_END_FBD_
(* the same logic as Structured Text *)
(* Network 1: Added by code generator *)
LonMaster(ptInData := ADR(InData_LON), ptOutData := ADR(OutData_LON), xRequestNeuronState := LonState, xResetNeuronState := LonReset);
GRU01.ModuleState := LonMaster.wModuleState;
(* Network 2 *)
Virtualfunctionalblock(bObjectIndex := 0, VT_Request := GRU01.NO_Request, VT_TimeSet := GRU01.NO_TimeSet, VT_AlarmSet := GRU01.NO_AlarmSet, VT_HCC1_ModeSet := GRU01.HCC1_ModeSet, VT_HCC1_TempSet := GRU01.HCC1_SetTemp, VT_HCC1_SuppTemp := GRU01.HCC1_SuppTemp, VT_HCC2_ModeSet := GRU01.HCC2_ModeSet, VT_HCC2_TempSet := GRU01.HCC2_SetTemp, VT_HCC2_SuppTemp := GRU01.HCC2_SuppTemp, VT_HCC3_ModeSet := GRU01.HCC3_ModeSet, VT_HCC3_TempSet := GRU01.HCC3_SetTemp, VT_HCC3_SuppTemp := GRU01.HCC3_SuppTemp, VT_DHW_ModeSet := GRU01.DHW_ModeSet, VT_DHW_SetPoint := GRU01.DHW_SetPoint, VT_CFD_SetEnable := GRU01.CFD_SetEnable, VT_CFD_SetMode := GRU01.CFD_SetMode, VT_CFD_SetPoint := GRU01.CFD_SetPoint, VT_BOC_SetEnable := GRU01.BOC_SetEnable, VT_BOC_SetMode := GRU01.BOC_SetMode, VT_BOC_SetPoint := GRU01.BOC_SetPoint);
GRU01.NO_Alarm := Virtualfunctionalblock.VT_Alarm;
GRU01.NO_RlyState := Virtualfunctionalblock.VT_RlyState;
GRU01.HCC1_SetMode := Virtualfunctionalblock.VT_HCC1_Mode;
GRU01.HCC1_SetTemp := Virtualfunctionalblock.VT_HCC1_Temp;
GRU01.HCC2_SetMode := Virtualfunctionalblock.VT_HCC2_Mode;
GRU01.HCC2_SetTemp := Virtualfunctionalblock.VT_HCC2_Temp;
GRU01.HCC3_SetMode := Virtualfunctionalblock.VT_HCC3_Mode;
GRU01.HCC3_SetTemp := Virtualfunctionalblock.VT_HCC3_Temp;
GRU01.DHW_ActTemp := Virtualfunctionalblock.VT_DHW_ActTemp;
GRU01.DHW_SetTemp := Virtualfunctionalblock.VT_DHW_TempSet;
GRU01.CFD_GetEnable := Virtualfunctionalblock.VT_CFD_GetEnable;
GRU01.CFD_Temp := Virtualfunctionalblock.VT_CFD_Temp;
GRU01.CFD_SetTemp := Virtualfunctionalblock.VT_CFD_SetTemp;
GRU01.BOC_GetEnable := Virtualfunctionalblock.VT_BOC_GetEnable;
GRU01.BOC_Temp := Virtualfunctionalblock.VT_BOC_Temp;
GRU01.BOC_SetTemp := Virtualfunctionalblock.VT_BOC_SetTemp;
GRU01.NO_Status := Virtualfunctionalblock.VT_Status;
END_PROGRAM

(* POU LON/Module_1/Master/Module_1_LonMaster, ST *)
FUNCTION_BLOCK Module_1_LonMaster
(******************************************)
(* Automatic generated code, do not edit! *)
(******************************************)
VAR_INPUT
	ptInData  : POINTER TO BYTE;
	ptOutData : POINTER TO BYTE;
	xRequestNeuronState : BOOL;
	xResetNeuronState : BOOL;
END_VAR
VAR_OUTPUT
	wModuleState : WORD; (* bit coded wModuleState:
	15: communication to I/O-module interrupted (error)
	14 - 08: reserved
	07: ready for Neuron initialization
	06: Neuron active
	05: user interface active
	04: internal module communication interrupted (error)
	03: CP synchronization running
	02: Neuron is configured online
	01 - 00: reserved *)

	typNeuronState : NeuronState;
	abNeuronId : ARRAY[0..5] OF BYTE;
	atypDomainData : ARRAY[0..1] OF DomainData;
	typApplicationMessage : ApplicationMessageData;
END_VAR
VAR
	bInternalCode : BYTE;
	bNvIndex : BYTE;
	wCpIndex : WORD;
	lonCom : FbLonBasicCommunication;

	xInitIsStarted : BOOL := FALSE;

	TimeoutTimer : TON;
	timeOutTime : TIME := T#1000ms;
	xStateMachineIsChecked : BOOL;
	xTimerStart : BOOL;

	iDomainTable : INT;
	xSendRequestPending : BOOL;
	trigRequest : R_TRIG;
	trigReset : R_TRIG;

	abMbxRxPrio0Buf: ARRAY [0..309] OF BYTE;
	abMbxRxPrio1Buf: ARRAY [0..517] OF BYTE;
	aMbxRxBufSize: ARRAY [0..1] OF UINT := 310, 518;
	aMbxRxBufList: ARRAY [0..1] OF POINTER TO BYTE;
	afbMbxRxFb: ARRAY [0..1] OF MBX2_RX_DEFRAG;
	astMbxRxCtx: ARRAY [0..1] OF stMbx2DefragContext;

	abMbxTxPrio0Buf: ARRAY [0..309] OF BYTE;
	abMbxTxPrio1Buf: ARRAY [0..517] OF BYTE;
	aMbxTxBufSize: ARRAY [0..1] OF UINT := 310, 518;
	aMbxTxBufList: ARRAY [0..1] OF POINTER TO BYTE;
	afbMbxTxFb: ARRAY [0..1] OF MBX2_TX_FRAG;

	astMbxTrackContext: ARRAY [0..0] OF stMbx2TrackContext;
END_VAR
VAR CONSTANT
END_VAR
aMbxRxBufList[0] := ADR(abMbxRxPrio0Buf[0]);
aMbxRxBufList[1] := ADR(abMbxRxPrio1Buf[0]);

aMbxTxBufList[0] := ADR(abMbxTxPrio0Buf[0]);
aMbxTxBufList[1] := ADR(abMbxTxPrio1Buf[0]);

mbxModule_1.Ressources.pDefragBufList := ADR(aMbxRxBufList);
mbxModule_1.Ressources.pDefragBufSizeList := ADR(aMbxRxBufSize);
mbxModule_1.Ressources.pDefragCtxPtrList := ADR(astMbxRxCtx);
mbxModule_1.Ressources.pDefragFbList := ADR(afbMbxRxFb);
mbxModule_1.Ressources.pFragBufList := ADR(aMbxTxBufList);
mbxModule_1.Ressources.pFragBufSizeList := ADR(aMbxTxBufSize);
mbxModule_1.Ressources.pFragFbList := ADR(afbMbxTxFb);

mbxModule_1.Ressources.unMaxAvailableRxPrioIndex := 1;
mbxModule_1.Ressources.unMaxAvailableTxPrioIndex := 1;

mbxModule_1.Ressources.pTrackStList := ADR(astMbxTrackContext);
mbxModule_1.Ressources.unMaxAvailableTrackIndex := 0;

mbxModule_1.Ressources.pabRxWin := ptInData + 1;
mbxModule_1.Ressources.pabTxWin := ptOutData + 1;
mbxModule_1.Ressources.bTxWinSize := 23;
mbxModule_1.Ressources.bRxWinSize := 23;

IF (mbxModule_1.bStatus.2 = TRUE) OR (mbxModule_1.bStatus.1 = TRUE) THEN
	mbxModule_1.MBX_RESET();
	xInitRunning_Module_1 := TRUE;
	xInitIsStarted := FALSE;
END_IF
mbxModule_1.MBX_CYCLE();

IF (mbxModule_1.bStatus.0 <> TRUE) THEN 
	wModuleState := 16#8000;
	RETURN;
ELSE
	wModuleState.15 := FALSE;
END_IF

xStateMachineIsChecked := FALSE;
IF xInitRunning_Module_1 = TRUE THEN
	IF xInitIsStarted = FALSE THEN
		SetParameter();
		lonCom.eInitState := INIT_SND_SGNTR_REQ;
		lonCom.CheckInitState();
		xInitIsStarted := TRUE;
		xStateMachineIsChecked := TRUE;
	END_IF
END_IF

typApplicationMessage.xMsgRcvd := FALSE;
typApplicationMessage.xRspRcvd := FALSE;
ResetNviUpdate();
WHILE (mbxModule_1.xRxPending) DO
	unLastLen_mbxModule_1 := mbxModule_1.unRxLen;
	mbxModule_1.pbRxData := ADR(InDataTelegram_Module_1);
	mbxModule_1.MBX_RETRIEVE();
	IF (mbxModule_1.nError <> MBX_OK) THEN EXIT; END_IF;
	bInternalCode := InDataTelegram_Module_1[0];

	IF (xInitRunning_Module_1 = TRUE) AND (lonCom.eInitState <> INIT_TRANSFER_CFG) THEN
		IF (FuCheckForValidInitCode(bInternalCode)) THEN
			SetParameter();
			lonCom.unLastLen := unLastLen_mbxModule_1;
			lonCom.CheckInitState();
			xInitRunning_Module_1 := NOT lonCom.xInitDone;
			xStateMachineIsChecked := TRUE;
		END_IF
	END_IF

	IF (bInternalCode = M2C_NVI_UPDT_OCCD) OR (bInternalCode = M2C_NV_VALUE_RSP) OR (bInternalCode = M2C_NVI_UPDT_TOUT) THEN
		bNvIndex := InDataTelegram_Module_1[1];
		CASE bNvIndex OF
			0, 2, 4: Module_1_PRG.SFPTnodeObject.DataReceived();
			6, 8, 10, 12, 14, 17, 19, 22, 24, 27, 29, 31, 33, 35, 37, 39, 41: Module_1_PRG.Virtualfunctionalblock.DataReceived();

		END_CASE;
	ELSIF (bInternalCode = M2C_CP_VALUE_RSP) THEN
		wCpIndex := InDataTelegram_Module_1[1] OR (InDataTelegram_Module_1[2] * 256);
		CASE wCpIndex OF

		END_CASE;
	ELSIF (bInternalCode = M2C_LON_MSG_RCVD) OR (bInternalCode = M2C_LON_RSP_RCVD) THEN
		ApplMsgReceived();
	ELSIF (bInternalCode = M2C_STATUS_RSP) THEN
		wModuleState := (wModuleState AND 16#FF00) + InDataTelegram_Module_1[1];
	ELSIF (bInternalCode = M2C_NEURON_ID) THEN
		FuMemCopy(ADR(InDataTelegram_Module_1[1]), ADR(abNeuronId), 6);
	ELSIF (bInternalCode = M2C_DOMAIN_DATA) THEN
		DomainDataRcvd();
	ELSIF (bInternalCode = M2C_MICRO_SERVER_STATUS_RSP) THEN
		NeuronStateRcvd();
	END_IF
END_WHILE

IF (xInitRunning_Module_1 = TRUE) AND ((lonCom.xCallStateMachine = TRUE) OR (TimeoutTimer.Q = TRUE)) AND (NOT xStateMachineIsChecked) THEN
	SetParameter();
	lonCom.xTimeOut := TimeoutTimer.Q;
	lonCom.CheckInitState();
END_IF
TimeoutTimer(IN:=lonCom.xTimerStart, PT:=timeOutTime);

trigRequest(CLK := xRequestNeuronState);
trigReset(CLK := xResetNeuronState);
IF (trigRequest.Q OR trigReset.Q) THEN
	RequestNeuronState();
END_IF
END_FUNCTION_BLOCK
ACTION ApplMsgReceived:
IF (InDataTelegram_Module_1[0] = M2C_LON_MSG_RCVD) THEN
	typApplicationMessage.typService := InDataTelegram_Module_1[1] AND 16#30;
	typApplicationMessage.bSourceSubnetId := InDataTelegram_Module_1[2];
	typApplicationMessage.bSourceNodeId := InDataTelegram_Module_1[3];
	typApplicationMessage.bCorrelator := InDataTelegram_Module_1[4];
	typApplicationMessage.bCode :=  InDataTelegram_Module_1[5];
	typApplicationMessage.bDataLength := UINT_TO_BYTE(unLastLen_mbxModule_1 - 6);
	IF typApplicationMessage.bDataLength > 48 THEN typApplicationMessage.bDataLength := 48; END_IF;
	FuMemSet(ADR(typApplicationMessage.abData), 0, SIZEOF(typApplicationMessage.abData));
	IF typApplicationMessage.bDataLength > 0 THEN
		FuMemCopy(ADR(InDataTelegram_Module_1[6]), ADR(typApplicationMessage.abData), typApplicationMessage.bDataLength);
	END_IF
	typApplicationMessage.xMsgRcvd := TRUE;
ELSE
	typApplicationMessage.typService := LON_RESPONSE;
	typApplicationMessage.bSourceSubnetId := InDataTelegram_Module_1[1];
	typApplicationMessage.bSourceNodeId := InDataTelegram_Module_1[2];
	typApplicationMessage.bCorrelator := 0;
	typApplicationMessage.bCode :=  InDataTelegram_Module_1[3];
	typApplicationMessage.bDataLength := UINT_TO_BYTE(unLastLen_mbxModule_1 - 4);
	IF typApplicationMessage.bDataLength > 48 THEN typApplicationMessage.bDataLength := 48; END_IF;
	FuMemSet(ADR(typApplicationMessage.abData), 0, SIZEOF(typApplicationMessage.abData));
	IF typApplicationMessage.bDataLength > 0 THEN
		FuMemCopy(ADR(InDataTelegram_Module_1[4]), ADR(typApplicationMessage.abData), typApplicationMessage.bDataLength);
	END_IF
	typApplicationMessage.xRspRcvd := TRUE;
END_IF
END_ACTION
ACTION DomainDataRcvd:
IF (unLastLen_mbxModule_1 = 17) THEN
	iDomainTable := InDataTelegram_Module_1[1];
	IF (iDomainTable < 0) OR (iDomainTable > 1) THEN RETURN; END_IF
	FuMemCopy(ADR(InDataTelegram_Module_1[2]), ADR(atypDomainData[iDomainTable].abDomainId), 6);
	atypDomainData[iDomainTable].bSubnet := InDataTelegram_Module_1[8];
	atypDomainData[iDomainTable].xIsNonClone := InDataTelegram_Module_1[9].7;
	atypDomainData[iDomainTable].bNodeId := InDataTelegram_Module_1[9] AND 16#7F;
	atypDomainData[iDomainTable].xIsInvalid := InDataTelegram_Module_1[10].7;
	atypDomainData[iDomainTable].bDomainIdLength := InDataTelegram_Module_1[10] AND 16#7F;
	FuMemCopy(ADR(InDataTelegram_Module_1[11]), ADR(atypDomainData[iDomainTable].abAuthenticationKey), 6);
END_IF
END_ACTION
ACTION NeuronStateRcvd:
IF (unLastLen_mbxModule_1 = 16) THEN
	typNeuronState.wCrcError := InDataTelegram_Module_1[1] + InDataTelegram_Module_1[2] * 256;
	typNeuronState.wTransactionTimeouts := InDataTelegram_Module_1[3] + InDataTelegram_Module_1[4] * 256;
	typNeuronState.wReceiveTransactionBuffersFull := InDataTelegram_Module_1[5] + InDataTelegram_Module_1[6] * 256;
	typNeuronState.wLostMessages := InDataTelegram_Module_1[7] + InDataTelegram_Module_1[8] * 256;
	typNeuronState.wMissedMessages := InDataTelegram_Module_1[9] + InDataTelegram_Module_1[10] * 256;
	typNeuronState.bResetCause := InDataTelegram_Module_1[11];
	typNeuronState.bNodeState := InDataTelegram_Module_1[12];
	typNeuronState.bFirmwareVersion := InDataTelegram_Module_1[13];
	typNeuronState.bLastErrorLogged := InDataTelegram_Module_1[14];
	typNeuronState.bModelNumber := InDataTelegram_Module_1[15];
END_IF
END_ACTION
ACTION RequestNeuronState:
OutDataTelegram_Module_1[0] := C2M_MICRO_SERVER_STATUS_QRY;
OutDataTelegram_Module_1[1] := BOOL_TO_BYTE(trigReset.Q);

mbxModule_1.bTxPrio := 1;
mbxModule_1.bTxProtID := 0;
mbxModule_1.pbTxData := ADR(OutDataTelegram_Module_1);
mbxModule_1.unTxLen := 2;
mbxModule_1.MBX_SEND();

IF (mbxModule_1.nError <> MBX_OK) THEN
	RETURN;
END_IF
END_ACTION
ACTION ResetNviUpdate:
Module_1_PRG.SFPTnodeObject.ResetNviUpdate();
Module_1_PRG.Virtualfunctionalblock.ResetNviUpdate();
END_ACTION
ACTION SetParameter:
lonCom.pMbx 			:= ADR(mbxModule_1);
lonCom.pInData 			:= ADR(InDataTelegram_Module_1);
lonCom.pOutData 		:= ADR(OutDataTelegram_Module_1);
lonCom.pTimer			:= ADR(TimeoutTimer);

lonCom.pActualSignature	:= ADR(abSignature_Module_1);
lonCom.pConfigBlock := ADR(abInterface_Module_1);
lonCom.wConfigSize 		:= wConfigSize_Module_1;
END_ACTION

(* POU LON/Module_1/NV_Interface/Module_1_SFPTnodeObject, ST *)
FUNCTION_BLOCK Module_1_SFPTnodeObject
(******************************************)
(* Automatic generated code, do not edit! *)
(******************************************)
VAR_INPUT
	bObjectIndex : BYTE := 0;
	nvoStatus : typSnvtObjStatus;
	nvoFileStat : typSnvtFileStatus;

END_VAR
VAR_OUTPUT
	nviRequest : typSnvtObjRequest;
	nviFileReq : typSnvtFileReq;
	nviFilePos : typSnvtFilePos;

END_VAR
VAR
	xSetOnce : BOOL := TRUE;
	xDataInUpdated : BOOL := FALSE;
	nvoStatusLast: typSnvtObjStatus;
	nvoFileStatLast: typSnvtFileStatus;

	cmd : BYTE;
	z : INT;
	bNvRelativeIdx : BYTE;
	bNvAbsoluteIdx : BYTE;
	wCpRelativeIdx : WORD;
	wCpAbsoluteIdx : WORD;
END_VAR
VAR CONSTANT
	bNvStartIndex : BYTE := 0;
	wCpStartIndex : WORD := 65535;
	bLmoCount : BYTE := 1;
END_VAR
IF (xInitRunning_Module_1 = TRUE) AND (xSetOnce = TRUE) THEN
	xSetOnce := FALSE;
	CachePointers();
	SetUpdateFlags();
END_IF

CheckUpdateFlags();
IF (xInitRunning_Module_1 = FALSE) AND (xDataInUpdated = FALSE) THEN
	IF (mbxModule_1.bStatus.0) THEN
		SendValueRequest();
	END_IF
END_IF

IF (xInitRunning_Module_1 = FALSE) AND (mbxModule_1.bStatus.0) THEN
	xSetOnce := TRUE;
	xDataInUpdated := FALSE;
	IF ((NOT FuMemCompare(ADR(nvoStatusLast), ADR(nvoStatus), ADR(nvoStatus.bStatusInformation) - ADR(nvoStatus))) OR (nvoStatus.bStatusInformation.7 = TRUE) OR (nvoStatusLast.bInternalUseOnly.1 = TRUE)) THEN
		FuSnvtObjStatusToRaw(ADR(nvoStatus), ADR(OutDataTelegram_Module_1[2]));

		bNvAbsoluteIdx := bNvStartIndex + bObjectIndex + (1 * bLmoCount);

		IF (FuDoNvoUpdate_Module_1(ADR(nvoStatus), ADR(nvoStatusLast), ADR(nvoStatus.bInternalUseOnly), ADR(nvoStatusLast.bInternalUseOnly), ADR(nvoStatus.bStatusInformation), bNvAbsoluteIdx, 6, SIZEOF(nvoStatus)) = FALSE) THEN
			RETURN;
		END_IF
	END_IF
	IF ((NOT FuMemCompare(ADR(nvoFileStatLast), ADR(nvoFileStat), ADR(nvoFileStat.bStatusInformation) - ADR(nvoFileStat))) OR (nvoFileStat.bStatusInformation.7 = TRUE) OR (nvoFileStatLast.bInternalUseOnly.1 = TRUE)) THEN
		FuSnvtFileStatusToRaw(ADR(nvoFileStat), ADR(OutDataTelegram_Module_1[2]));

		bNvAbsoluteIdx := bNvStartIndex + bObjectIndex + (3 * bLmoCount);

		IF (FuDoNvoUpdate_Module_1(ADR(nvoFileStat), ADR(nvoFileStatLast), ADR(nvoFileStat.bInternalUseOnly), ADR(nvoFileStatLast.bInternalUseOnly), ADR(nvoFileStat.bStatusInformation), bNvAbsoluteIdx, 27, SIZEOF(nvoFileStat)) = FALSE) THEN
			RETURN;
		END_IF
	END_IF

END_IF
END_FUNCTION_BLOCK
ACTION CachePointers:
;
END_ACTION
ACTION CheckUpdateFlags:
xDataInUpdated := (NOT nviRequest.bInternalUseOnly.0) AND (NOT nviFileReq.bInternalUseOnly.0) AND (NOT nviFilePos.bInternalUseOnly.0) AND TRUE;
END_ACTION
ACTION DataReceived:
cmd := InDataTelegram_Module_1[0];
IF (cmd = M2C_NVI_UPDT_OCCD) OR (cmd = M2C_NV_VALUE_RSP) OR (cmd = M2C_NVI_UPDT_TOUT) THEN
	bNvRelativeIdx := (InDataTelegram_Module_1[1] - bNvStartIndex - bObjectIndex) / bLmoCount;
	CASE bNvRelativeIdx OF
	0:
		IF (cmd = M2C_NVI_UPDT_OCCD) OR (cmd = M2C_NV_VALUE_RSP) THEN
			IF (unLastLen_mbxModule_1 = (2 + 3)) THEN
				FuRawToSnvtObjRequest(ADR(InDataTelegram_Module_1[2]), ADR(nviRequest));
				nviRequest.bInternalUseOnly.0 := FALSE;
				nviRequest.bStatusInformation := FuInkrementNviStatus(nviRequest.bStatusInformation);
			ELSIF (unLastLen_mbxModule_1 = 2) THEN
				nviRequest.bStatusInformation := FuInkrementNviStatus(nviRequest.bStatusInformation);
			END_IF
		ELSIF (cmd = M2C_NVI_UPDT_TOUT) THEN
			IF (unLastLen_mbxModule_1 = 3) THEN
				nviRequest.bStatusInformation.4 := BYTE_TO_BOOL(InDataTelegram_Module_1[2]);
			END_IF
		END_IF
	2:
		IF (cmd = M2C_NVI_UPDT_OCCD) OR (cmd = M2C_NV_VALUE_RSP) THEN
			IF (unLastLen_mbxModule_1 = (2 + 12)) THEN
				FuRawToSnvtFileReq(ADR(InDataTelegram_Module_1[2]), ADR(nviFileReq));
				nviFileReq.bInternalUseOnly.0 := FALSE;
				nviFileReq.bStatusInformation := FuInkrementNviStatus(nviFileReq.bStatusInformation);
			ELSIF (unLastLen_mbxModule_1 = 2) THEN
				nviFileReq.bStatusInformation := FuInkrementNviStatus(nviFileReq.bStatusInformation);
			END_IF
		ELSIF (cmd = M2C_NVI_UPDT_TOUT) THEN
			IF (unLastLen_mbxModule_1 = 3) THEN
				nviFileReq.bStatusInformation.4 := BYTE_TO_BOOL(InDataTelegram_Module_1[2]);
			END_IF
		END_IF
	4:
		IF (cmd = M2C_NVI_UPDT_OCCD) OR (cmd = M2C_NV_VALUE_RSP) THEN
			IF (unLastLen_mbxModule_1 = (2 + 6)) THEN
				FuRawToSnvtFilePos(ADR(InDataTelegram_Module_1[2]), ADR(nviFilePos));
				nviFilePos.bInternalUseOnly.0 := FALSE;
				nviFilePos.bStatusInformation := FuInkrementNviStatus(nviFilePos.bStatusInformation);
			ELSIF (unLastLen_mbxModule_1 = 2) THEN
				nviFilePos.bStatusInformation := FuInkrementNviStatus(nviFilePos.bStatusInformation);
			END_IF
		ELSIF (cmd = M2C_NVI_UPDT_TOUT) THEN
			IF (unLastLen_mbxModule_1 = 3) THEN
				nviFilePos.bStatusInformation.4 := BYTE_TO_BOOL(InDataTelegram_Module_1[2]);
			END_IF
		END_IF

	END_CASE
ELSIF (cmd = M2C_CP_VALUE_RSP) THEN
	wCpRelativeIdx := ((InDataTelegram_Module_1[1] + InDataTelegram_Module_1[2] * 256) - wCpStartIndex - bObjectIndex) / bLmoCount;
	CASE wCpRelativeIdx OF

	END_CASE
END_IF
END_ACTION
ACTION ResetNviUpdate:
nviRequest.bStatusInformation := nviRequest.bStatusInformation AND 16#F8;
nviFileReq.bStatusInformation := nviFileReq.bStatusInformation AND 16#F8;
nviFilePos.bStatusInformation := nviFilePos.bStatusInformation AND 16#F8;
;
END_ACTION
ACTION SendValueRequest:
IF (FuSendNviValueReq_Module_1(ADR(nviRequest.bInternalUseOnly), bNvStartIndex + bObjectIndex + (0 * bLmoCount)) = FALSE) THEN
	RETURN;
END_IF

IF (FuSendNviValueReq_Module_1(ADR(nviFileReq.bInternalUseOnly), bNvStartIndex + bObjectIndex + (2 * bLmoCount)) = FALSE) THEN
	RETURN;
END_IF

IF (FuSendNviValueReq_Module_1(ADR(nviFilePos.bInternalUseOnly), bNvStartIndex + bObjectIndex + (4 * bLmoCount)) = FALSE) THEN
	RETURN;
END_IF

;
END_ACTION
ACTION SetUpdateFlags:
nviRequest.bInternaluseOnly.0 := TRUE;
nvoStatusLast.bInternaluseOnly.1 := TRUE;
nvoStatusLast.bInternaluseOnly.7 := FALSE;
nviFileReq.bInternaluseOnly.0 := TRUE;
nvoFileStatLast.bInternaluseOnly.1 := TRUE;
nvoFileStatLast.bInternaluseOnly.7 := FALSE;
nviFilePos.bInternaluseOnly.0 := TRUE;
;
END_ACTION

(* POU LON/Shared/Internal/FuSnvtObjStatusToRaw, ST *)
FUNCTION FuSnvtObjStatusToRaw : BOOL
(******************************************)
(* Automatic generated code, do not edit! *)
(******************************************)
VAR_INPUT
	NvDataIn :  POINTER TO typSnvtObjStatus;
	DataOut : POINTER TO ARRAY[0..5] OF BYTE;
END_VAR
VAR
END_VAR
DataOut^[0] := WORD_TO_BYTE(SHR(NvDataIn^.wObjectId, 8));
DataOut^[1] := WORD_TO_BYTE(NvDataIn^.wObjectId);

DataOut^[2] := NvDataIn^.bBitfieldByteOffset2;

DataOut^[3] := NvDataIn^.bBitfieldByteOffset3;

DataOut^[4] := NvDataIn^.bBitfieldByteOffset4;

DataOut^[5] := NvDataIn^.bBitfieldByteOffset5;

FuSnvtObjStatusToRaw := TRUE;
END_FUNCTION

(* POU LON/Module_1/Internal/FuDoNvoUpdate_Module_1, ST *)
FUNCTION FuDoNvoUpdate_Module_1 : BOOL
(******************************************)
(* Automatic generated code, do not edit! *)
(******************************************)
VAR_INPUT
	ptNvo : POINTER TO BYTE;
	ptNvoLast : POINTER TO BYTE;
	ptNvoInternalUse : POINTER TO BYTE;
	ptNvoLastInternalUse : POINTER TO BYTE;
	ptNvoStatusInformation : POINTER TO BYTE;
	bNvoIndex : BYTE;
	uiNvoLength : UINT;
	uiNvoVariableLength : UINT;
END_VAR
IF (ptNvoLastInternalUse^.1 = TRUE) AND (ptNvoStatusInformation^.7 = FALSE) THEN
	OutDataTelegram_Module_1[0] := C2M_NV_VALUE;
ELSE
	OutDataTelegram_Module_1[0] := C2M_NVO_PROPAGATE;
END_IF
OutDataTelegram_Module_1[1] := bNvoIndex;

mbxModule_1.bTxPrio := BOOL_TO_BYTE(ptNvoLastInternalUse^.7);
mbxModule_1.bTxProtID := 0;
mbxModule_1.pbTxData := ADR(OutDataTelegram_Module_1);
mbxModule_1.unTxLen := 2 + uiNvoLength;
mbxModule_1.MBX_SEND();

IF (mbxModule_1.nError <> MBX_OK) THEN
	FuDoNvoUpdate_Module_1 := FALSE;
	RETURN;
END_IF

ptNvoLastInternalUse^.1 := FALSE;
ptNvoInternalUse^ := ptNvoLastInternalUse^;
FuMemCopy(ptNvo, ptNvoLast, uiNvoVariableLength);

FuDoNvoUpdate_Module_1 := TRUE;
END_FUNCTION

(* POU LON/Shared/Internal/FuSnvtFileStatusToRaw, ST *)
FUNCTION FuSnvtFileStatusToRaw : BOOL
(******************************************)
(* Automatic generated code, do not edit! *)
(******************************************)
VAR_INPUT
	NvDataIn :  POINTER TO typSnvtFileStatus;
	DataOut : POINTER TO ARRAY[0..26] OF BYTE;
END_VAR
VAR
END_VAR
DataOut^[0] := NvDataIn^.bStatus;

DataOut^[1] := WORD_TO_BYTE(SHR(NvDataIn^.wNumberOfFiles, 8));
DataOut^[2] := WORD_TO_BYTE(NvDataIn^.wNumberOfFiles);

DataOut^[3] := WORD_TO_BYTE(SHR(NvDataIn^.wSelectedFile, 8));
DataOut^[4] := WORD_TO_BYTE(NvDataIn^.wSelectedFile);

DataOut^[5] := NvDataIn^.abAdr[0];
DataOut^[6] := NvDataIn^.abAdr[1];
DataOut^[7] := NvDataIn^.abAdr[2];
DataOut^[8] := NvDataIn^.abAdr[3];
DataOut^[9] := NvDataIn^.abAdr[4];
DataOut^[10] := NvDataIn^.abAdr[5];
DataOut^[11] := NvDataIn^.abAdr[6];
DataOut^[12] := NvDataIn^.abAdr[7];
DataOut^[13] := NvDataIn^.abAdr[8];
DataOut^[14] := NvDataIn^.abAdr[9];
DataOut^[15] := NvDataIn^.abAdr[10];
DataOut^[16] := NvDataIn^.abAdr[11];
DataOut^[17] := NvDataIn^.abAdr[12];
DataOut^[18] := NvDataIn^.abAdr[13];
DataOut^[19] := NvDataIn^.abAdr[14];
DataOut^[20] := NvDataIn^.abAdr[15];
DataOut^[21] := NvDataIn^.abAdr[16];
DataOut^[22] := NvDataIn^.abAdr[17];
DataOut^[23] := NvDataIn^.abAdr[18];
DataOut^[24] := NvDataIn^.abAdr[19];
DataOut^[25] := NvDataIn^.abAdr[20];
DataOut^[26] := NvDataIn^.abAdr[21];

FuSnvtFileStatusToRaw := TRUE;
END_FUNCTION

(* POU LON/Module_1/Internal/FuSendNviValueReq_Module_1, ST *)
FUNCTION FuSendNviValueReq_Module_1 : BOOL
(******************************************)
(* Automatic generated code, do not edit! *)
(******************************************)
VAR_INPUT
	ptInternalUseOnly : POINTER TO BYTE;
	bNvIndex : BYTE;
END_VAR
IF ptInternalUseOnly^.0 = TRUE THEN
	OutDataTelegram_Module_1[0] := C2M_NV_VALUE_QRY;
	OutDataTelegram_Module_1[1] := bNvIndex;

	mbxModule_1.bTxPrio := 1;
	mbxModule_1.bTxProtID := 0;
	mbxModule_1.pbTxData := ADR(OutDataTelegram_Module_1);
	mbxModule_1.unTxLen := 2;
	mbxModule_1.MBX_SEND();

	IF (mbxModule_1.nError <> MBX_OK) THEN
		FuSendNviValueReq_Module_1 := FALSE;
		RETURN;
	END_IF
	ptInternalUseOnly^.0 := FALSE;
END_IF

FuSendNviValueReq_Module_1 := TRUE;
END_FUNCTION

(* POU LON/Module_1/NV_Interface/Module_1_Virtualfunctionalblock, ST *)
FUNCTION_BLOCK Module_1_Virtualfunctionalblock
(******************************************)
(* Automatic generated code, do not edit! *)
(******************************************)
VAR_INPUT
	bObjectIndex : BYTE := 0;
	VT_Request : typSnvtObjRequest;
	VT_TimeSet : typSnvtTimeStamp;
	VT_AlarmSet : typSnvtAlarm;
	VT_HCC1_ModeSet : typSnvtHvacMode;
	VT_HCC1_TempSet : typSnvtTempP;
	VT_HCC1_SuppTemp : typSnvtTempP;
	VT_HCC2_ModeSet : typSnvtHvacMode;
	VT_HCC2_TempSet : typSnvtTempP;
	VT_HCC2_SuppTemp : typSnvtTempP;
	VT_HCC3_ModeSet : typSnvtHvacMode;
	VT_HCC3_TempSet : typSnvtTempP;
	VT_HCC3_SuppTemp : typSnvtTempP;
	VT_DHW_ModeSet : typSnvtHvacMode;
	VT_DHW_SetPoint : typSnvtTempP;
	VT_CFD_SetEnable : typSnvtSwitch;
	VT_CFD_SetMode : typSnvtHvacMode;
	VT_CFD_SetPoint : typSnvtTempP;
	VT_BOC_SetEnable : typSnvtSwitch;
	VT_BOC_SetMode : typSnvtHvacMode;
	VT_BOC_SetPoint : typSnvtTempP;

END_VAR
VAR_OUTPUT
	VT_Status : typSnvtObjStatus;
	VT_Alarm : typSnvtAlarm;
	VT_RlyState : typSnvtState;
	VT_HCC1_Mode : typSnvtHvacMode;
	VT_HCC1_Temp : typSnvtTempP;
	VT_HCC2_Mode : typSnvtHvacMode;
	VT_HCC2_Temp : typSnvtTempP;
	VT_HCC3_Mode : typSnvtHvacMode;
	VT_HCC3_Temp : typSnvtTempP;
	VT_DHW_ActTemp : typSnvtTempP;
	VT_DHW_TempSet : typSnvtTempP;
	VT_CFD_GetEnable : typSnvtSwitch;
	VT_CFD_Temp : typSnvtTempP;
	VT_CFD_SetTemp : typSnvtTempP;
	VT_BOC_GetEnable : typSnvtSwitch;
	VT_BOC_Temp : typSnvtTempP;
	VT_BOC_SetTemp : typSnvtTempP;

END_VAR
VAR
	xSetOnce : BOOL := TRUE;
	xDataInUpdated : BOOL := FALSE;
	VT_RequestLast: typSnvtObjRequest;
	VT_TimeSetLast: typSnvtTimeStamp;
	VT_AlarmSetLast: typSnvtAlarm;
	paNviSnvtHvacMode : ARRAY[0..2] OF POINTER TO typSnvtHvacMode;
	aNviSnvtHvacModeIndex : ARRAY[0..2] OF BYTE := 7,12,17;
	paNviSnvtTempP : ARRAY[0..8] OF POINTER TO typSnvtTempP;
	aNviSnvtTempPIndex : ARRAY[0..8] OF BYTE := 9,14,19,22,24,28,30,34,36;
	paNviSnvtSwitch : ARRAY[0..1] OF POINTER TO typSnvtSwitch;
	aNviSnvtSwitchIndex : ARRAY[0..1] OF BYTE := 26,32;
	paNvoSnvtHvacMode : ARRAY[0..5] OF POINTER TO typSnvtHvacMode;
	aNvoSnvtHvacModeIndex : ARRAY[0..5] OF BYTE := 6,11,16,21,27,33;
	aNvoSnvtHvacModeLast : ARRAY[0..5] OF typSnvtHvacMode;
	aNvoSnvtHvacModePriority : ARRAY[0..0] OF BYTE := 16#00;
	paNvoSnvtTempP : ARRAY[0..8] OF POINTER TO typSnvtTempP;
	aNvoSnvtTempPIndex : ARRAY[0..8] OF BYTE := 8,10,13,15,18,20,23,29,35;
	aNvoSnvtTempPLast : ARRAY[0..8] OF typSnvtTempP;
	aNvoSnvtTempPPriority : ARRAY[0..1] OF BYTE := 16#00, 16#00;
	paNvoSnvtSwitch : ARRAY[0..1] OF POINTER TO typSnvtSwitch;
	aNvoSnvtSwitchIndex : ARRAY[0..1] OF BYTE := 25,31;
	aNvoSnvtSwitchLast : ARRAY[0..1] OF typSnvtSwitch;
	aNvoSnvtSwitchPriority : ARRAY[0..0] OF BYTE := 16#00;

	cmd : BYTE;
	z : INT;
	bNvRelativeIdx : BYTE;
	bNvAbsoluteIdx : BYTE;
	wCpRelativeIdx : WORD;
	wCpAbsoluteIdx : WORD;
END_VAR
VAR CONSTANT
	bNvStartIndex : BYTE := 5;
	wCpStartIndex : WORD := 65535;
	bLmoCount : BYTE := 1;
END_VAR
IF (xInitRunning_Module_1 = TRUE) AND (xSetOnce = TRUE) THEN
	xSetOnce := FALSE;
	CachePointers();
	SetUpdateFlags();
END_IF

CheckUpdateFlags();
IF (xInitRunning_Module_1 = FALSE) AND (xDataInUpdated = FALSE) THEN
	IF (mbxModule_1.bStatus.0) THEN
		SendValueRequest();
	END_IF
END_IF

IF (xInitRunning_Module_1 = FALSE) AND (mbxModule_1.bStatus.0) THEN
	xSetOnce := TRUE;
	xDataInUpdated := FALSE;
	IF ((NOT FuMemCompare(ADR(VT_RequestLast), ADR(VT_Request), ADR(VT_Request.bStatusInformation) - ADR(VT_Request))) OR (VT_Request.bStatusInformation.7 = TRUE) OR (VT_RequestLast.bInternalUseOnly.1 = TRUE)) THEN
		FuSnvtObjRequestToRaw(ADR(VT_Request), ADR(OutDataTelegram_Module_1[2]));

		bNvAbsoluteIdx := bNvStartIndex + bObjectIndex + (0 * bLmoCount);

		IF (FuDoNvoUpdate_Module_1(ADR(VT_Request), ADR(VT_RequestLast), ADR(VT_Request.bInternalUseOnly), ADR(VT_RequestLast.bInternalUseOnly), ADR(VT_Request.bStatusInformation), bNvAbsoluteIdx, 3, SIZEOF(VT_Request)) = FALSE) THEN
			RETURN;
		END_IF
	END_IF
	IF ((NOT FuMemCompare(ADR(VT_TimeSetLast), ADR(VT_TimeSet), ADR(VT_TimeSet.bStatusInformation) - ADR(VT_TimeSet))) OR (VT_TimeSet.bStatusInformation.7 = TRUE) OR (VT_TimeSetLast.bInternalUseOnly.1 = TRUE)) THEN
		FuSnvtTimeStampToRaw(ADR(VT_TimeSet), ADR(OutDataTelegram_Module_1[2]));

		bNvAbsoluteIdx := bNvStartIndex + bObjectIndex + (2 * bLmoCount);

		IF (FuDoNvoUpdate_Module_1(ADR(VT_TimeSet), ADR(VT_TimeSetLast), ADR(VT_TimeSet.bInternalUseOnly), ADR(VT_TimeSetLast.bInternalUseOnly), ADR(VT_TimeSet.bStatusInformation), bNvAbsoluteIdx, 7, SIZEOF(VT_TimeSet)) = FALSE) THEN
			RETURN;
		END_IF
	END_IF
	IF ((NOT FuMemCompare(ADR(VT_AlarmSetLast), ADR(VT_AlarmSet), ADR(VT_AlarmSet.bStatusInformation) - ADR(VT_AlarmSet))) OR (VT_AlarmSet.bStatusInformation.7 = TRUE) OR (VT_AlarmSetLast.bInternalUseOnly.1 = TRUE)) THEN
		FuSnvtAlarmToRaw(ADR(VT_AlarmSet), ADR(OutDataTelegram_Module_1[2]));

		bNvAbsoluteIdx := bNvStartIndex + bObjectIndex + (4 * bLmoCount);

		IF (FuDoNvoUpdate_Module_1(ADR(VT_AlarmSet), ADR(VT_AlarmSetLast), ADR(VT_AlarmSet.bInternalUseOnly), ADR(VT_AlarmSetLast.bInternalUseOnly), ADR(VT_AlarmSet.bStatusInformation), bNvAbsoluteIdx, 29, SIZEOF(VT_AlarmSet)) = FALSE) THEN
			RETURN;
		END_IF
	END_IF
	FOR z := 0 TO 5 DO
		IF ((NOT FuMemCompare(ADR(aNvoSnvtHvacModeLast[z]), paNvoSnvtHvacMode[z], ADR(paNvoSnvtHvacMode[z]^.bStatusInformation) - paNvoSnvtHvacMode[z])) OR (paNvoSnvtHvacMode[z]^.bStatusInformation.7 = TRUE) OR (aNvoSnvtHvacModeLast[z].bInternalUseOnly.1 = TRUE)) THEN
			FuSnvtHvacModeToRaw(paNvoSnvtHvacMode[z], ADR(OutDataTelegram_Module_1[2]));

			bNvAbsoluteIdx := bNvStartIndex + bObjectIndex + (aNvoSnvtHvacModeIndex[z] * bLmoCount);

			IF (FuDoNvoUpdate_Module_1(paNvoSnvtHvacMode[z], ADR(aNvoSnvtHvacModeLast[z]), ADR(paNvoSnvtHvacMode[z]^.bInternalUseOnly), ADR(aNvoSnvtHvacModeLast[z].bInternalUseOnly), ADR(paNvoSnvtHvacMode[z]^.bStatusInformation), bNvAbsoluteIdx, 1, SIZEOF(aNvoSnvtHvacModeLast[z])) = FALSE) THEN
				RETURN;
			END_IF
		END_IF
	END_FOR
	FOR z := 0 TO 8 DO
		IF ((NOT FuMemCompare(ADR(aNvoSnvtTempPLast[z]), paNvoSnvtTempP[z], ADR(paNvoSnvtTempP[z]^.bStatusInformation) - paNvoSnvtTempP[z])) OR (paNvoSnvtTempP[z]^.bStatusInformation.7 = TRUE) OR (aNvoSnvtTempPLast[z].bInternalUseOnly.1 = TRUE)) THEN
			FuSnvtTempPToRaw(paNvoSnvtTempP[z], ADR(OutDataTelegram_Module_1[2]));

			bNvAbsoluteIdx := bNvStartIndex + bObjectIndex + (aNvoSnvtTempPIndex[z] * bLmoCount);

			IF (FuDoNvoUpdate_Module_1(paNvoSnvtTempP[z], ADR(aNvoSnvtTempPLast[z]), ADR(paNvoSnvtTempP[z]^.bInternalUseOnly), ADR(aNvoSnvtTempPLast[z].bInternalUseOnly), ADR(paNvoSnvtTempP[z]^.bStatusInformation), bNvAbsoluteIdx, 2, SIZEOF(aNvoSnvtTempPLast[z])) = FALSE) THEN
				RETURN;
			END_IF
		END_IF
	END_FOR
	FOR z := 0 TO 1 DO
		IF ((NOT FuMemCompare(ADR(aNvoSnvtSwitchLast[z]), paNvoSnvtSwitch[z], ADR(paNvoSnvtSwitch[z]^.bStatusInformation) - paNvoSnvtSwitch[z])) OR (paNvoSnvtSwitch[z]^.bStatusInformation.7 = TRUE) OR (aNvoSnvtSwitchLast[z].bInternalUseOnly.1 = TRUE)) THEN
			FuSnvtSwitchToRaw(paNvoSnvtSwitch[z], ADR(OutDataTelegram_Module_1[2]));

			bNvAbsoluteIdx := bNvStartIndex + bObjectIndex + (aNvoSnvtSwitchIndex[z] * bLmoCount);

			IF (FuDoNvoUpdate_Module_1(paNvoSnvtSwitch[z], ADR(aNvoSnvtSwitchLast[z]), ADR(paNvoSnvtSwitch[z]^.bInternalUseOnly), ADR(aNvoSnvtSwitchLast[z].bInternalUseOnly), ADR(paNvoSnvtSwitch[z]^.bStatusInformation), bNvAbsoluteIdx, 2, SIZEOF(aNvoSnvtSwitchLast[z])) = FALSE) THEN
				RETURN;
			END_IF
		END_IF
	END_FOR

END_IF
END_FUNCTION_BLOCK
ACTION CachePointers:
paNviSnvtHvacMode[0] := ADR(VT_HCC1_Mode);
paNviSnvtHvacMode[1] := ADR(VT_HCC2_Mode);
paNviSnvtHvacMode[2] := ADR(VT_HCC3_Mode);
paNviSnvtTempP[0] := ADR(VT_HCC1_Temp);
paNviSnvtTempP[1] := ADR(VT_HCC2_Temp);
paNviSnvtTempP[2] := ADR(VT_HCC3_Temp);
paNviSnvtTempP[3] := ADR(VT_DHW_ActTemp);
paNviSnvtTempP[4] := ADR(VT_DHW_TempSet);
paNviSnvtTempP[5] := ADR(VT_CFD_Temp);
paNviSnvtTempP[6] := ADR(VT_CFD_SetTemp);
paNviSnvtTempP[7] := ADR(VT_BOC_Temp);
paNviSnvtTempP[8] := ADR(VT_BOC_SetTemp);
paNviSnvtSwitch[0] := ADR(VT_CFD_GetEnable);
paNviSnvtSwitch[1] := ADR(VT_BOC_GetEnable);
paNvoSnvtHvacMode[0] := ADR(VT_HCC1_ModeSet);
paNvoSnvtHvacMode[1] := ADR(VT_HCC2_ModeSet);
paNvoSnvtHvacMode[2] := ADR(VT_HCC3_ModeSet);
paNvoSnvtHvacMode[3] := ADR(VT_DHW_ModeSet);
paNvoSnvtHvacMode[4] := ADR(VT_CFD_SetMode);
paNvoSnvtHvacMode[5] := ADR(VT_BOC_SetMode);
paNvoSnvtTempP[0] := ADR(VT_HCC1_TempSet);
paNvoSnvtTempP[1] := ADR(VT_HCC1_SuppTemp);
paNvoSnvtTempP[2] := ADR(VT_HCC2_TempSet);
paNvoSnvtTempP[3] := ADR(VT_HCC2_SuppTemp);
paNvoSnvtTempP[4] := ADR(VT_HCC3_TempSet);
paNvoSnvtTempP[5] := ADR(VT_HCC3_SuppTemp);
paNvoSnvtTempP[6] := ADR(VT_DHW_SetPoint);
paNvoSnvtTempP[7] := ADR(VT_CFD_SetPoint);
paNvoSnvtTempP[8] := ADR(VT_BOC_SetPoint);
paNvoSnvtSwitch[0] := ADR(VT_CFD_SetEnable);
paNvoSnvtSwitch[1] := ADR(VT_BOC_SetEnable);
;
END_ACTION
ACTION CheckUpdateFlags:
xDataInUpdated := (NOT VT_Status.bInternalUseOnly.0) AND (NOT VT_Alarm.bInternalUseOnly.0) AND (NOT VT_RlyState.bInternalUseOnly.0) AND TRUE;
FOR z := 0 TO 2 DO
	xDataInUpdated := xDataInUpdated AND (NOT paNviSnvtHvacMode[z]^.bInternalUseOnly.0);
END_FOR
FOR z := 0 TO 8 DO
	xDataInUpdated := xDataInUpdated AND (NOT paNviSnvtTempP[z]^.bInternalUseOnly.0);
END_FOR
FOR z := 0 TO 1 DO
	xDataInUpdated := xDataInUpdated AND (NOT paNviSnvtSwitch[z]^.bInternalUseOnly.0);
END_FOR
END_ACTION
ACTION DataReceived:
cmd := InDataTelegram_Module_1[0];
IF (cmd = M2C_NVI_UPDT_OCCD) OR (cmd = M2C_NV_VALUE_RSP) OR (cmd = M2C_NVI_UPDT_TOUT) THEN
	bNvRelativeIdx := (InDataTelegram_Module_1[1] - bNvStartIndex - bObjectIndex) / bLmoCount;
	CASE bNvRelativeIdx OF
	1:
		IF (cmd = M2C_NVI_UPDT_OCCD) OR (cmd = M2C_NV_VALUE_RSP) THEN
			IF (unLastLen_mbxModule_1 = (2 + 6)) THEN
				FuRawToSnvtObjStatus(ADR(InDataTelegram_Module_1[2]), ADR(VT_Status));
				VT_Status.bInternalUseOnly.0 := FALSE;
				VT_Status.bStatusInformation := FuInkrementNviStatus(VT_Status.bStatusInformation);
			ELSIF (unLastLen_mbxModule_1 = 2) THEN
				VT_Status.bStatusInformation := FuInkrementNviStatus(VT_Status.bStatusInformation);
			END_IF
		ELSIF (cmd = M2C_NVI_UPDT_TOUT) THEN
			IF (unLastLen_mbxModule_1 = 3) THEN
				VT_Status.bStatusInformation.4 := BYTE_TO_BOOL(InDataTelegram_Module_1[2]);
			END_IF
		END_IF
	3:
		IF (cmd = M2C_NVI_UPDT_OCCD) OR (cmd = M2C_NV_VALUE_RSP) THEN
			IF (unLastLen_mbxModule_1 = (2 + 29)) THEN
				FuRawToSnvtAlarm(ADR(InDataTelegram_Module_1[2]), ADR(VT_Alarm));
				VT_Alarm.bInternalUseOnly.0 := FALSE;
				VT_Alarm.bStatusInformation := FuInkrementNviStatus(VT_Alarm.bStatusInformation);
			ELSIF (unLastLen_mbxModule_1 = 2) THEN
				VT_Alarm.bStatusInformation := FuInkrementNviStatus(VT_Alarm.bStatusInformation);
			END_IF
		ELSIF (cmd = M2C_NVI_UPDT_TOUT) THEN
			IF (unLastLen_mbxModule_1 = 3) THEN
				VT_Alarm.bStatusInformation.4 := BYTE_TO_BOOL(InDataTelegram_Module_1[2]);
			END_IF
		END_IF
	5:
		IF (cmd = M2C_NVI_UPDT_OCCD) OR (cmd = M2C_NV_VALUE_RSP) THEN
			IF (unLastLen_mbxModule_1 = (2 + 2)) THEN
				FuRawToSnvtState(ADR(InDataTelegram_Module_1[2]), ADR(VT_RlyState));
				VT_RlyState.bInternalUseOnly.0 := FALSE;
				VT_RlyState.bStatusInformation := FuInkrementNviStatus(VT_RlyState.bStatusInformation);
			ELSIF (unLastLen_mbxModule_1 = 2) THEN
				VT_RlyState.bStatusInformation := FuInkrementNviStatus(VT_RlyState.bStatusInformation);
			END_IF
		ELSIF (cmd = M2C_NVI_UPDT_TOUT) THEN
			IF (unLastLen_mbxModule_1 = 3) THEN
				VT_RlyState.bStatusInformation.4 := BYTE_TO_BOOL(InDataTelegram_Module_1[2]);
			END_IF
		END_IF
	7, 12, 17:
		IF (cmd = M2C_NVI_UPDT_OCCD) OR (cmd = M2C_NV_VALUE_RSP) THEN
			IF (unLastLen_mbxModule_1 = (2 + 1)) THEN
				FOR z := 0 TO 2 DO
					IF aNviSnvtHvacModeIndex[z] = bNvRelativeIdx THEN
						FuRawToSnvtHvacMode(ADR(InDataTelegram_Module_1[2]), paNviSnvtHvacMode[z]);
						paNviSnvtHvacMode[z]^.bInternalUseOnly.0 := FALSE;
						paNviSnvtHvacMode[z]^.bStatusInformation := FuInkrementNviStatus(paNviSnvtHvacMode[z]^.bStatusInformation);
						EXIT;
					END_IF
				END_FOR
			ELSIF (unLastLen_mbxModule_1 = 2) THEN
				FOR z := 0 TO 2 DO
					IF aNviSnvtHvacModeIndex[z] = bNvRelativeIdx THEN
						paNviSnvtHvacMode[z]^.bStatusInformation := FuInkrementNviStatus(paNviSnvtHvacMode[z]^.bStatusInformation);
						EXIT;
					END_IF
				END_FOR
			END_IF
		ELSIF (cmd = M2C_NVI_UPDT_TOUT) THEN
			IF (unLastLen_mbxModule_1 = 3) THEN
				FOR z := 0 TO 2 DO
					IF aNviSnvtHvacModeIndex[z] = bNvRelativeIdx THEN
						paNviSnvtHvacMode[z]^.bStatusInformation.4 := BYTE_TO_BOOL(InDataTelegram_Module_1[2]);
						EXIT;
					END_IF
				END_FOR
			END_IF
		END_IF
	9, 14, 19, 22, 24, 28, 30, 34, 36:
		IF (cmd = M2C_NVI_UPDT_OCCD) OR (cmd = M2C_NV_VALUE_RSP) THEN
			IF (unLastLen_mbxModule_1 = (2 + 2)) THEN
				FOR z := 0 TO 8 DO
					IF aNviSnvtTempPIndex[z] = bNvRelativeIdx THEN
						FuRawToSnvtTempP(ADR(InDataTelegram_Module_1[2]), paNviSnvtTempP[z]);
						paNviSnvtTempP[z]^.bInternalUseOnly.0 := FALSE;
						paNviSnvtTempP[z]^.bStatusInformation := FuInkrementNviStatus(paNviSnvtTempP[z]^.bStatusInformation);
						EXIT;
					END_IF
				END_FOR
			ELSIF (unLastLen_mbxModule_1 = 2) THEN
				FOR z := 0 TO 8 DO
					IF aNviSnvtTempPIndex[z] = bNvRelativeIdx THEN
						paNviSnvtTempP[z]^.bStatusInformation := FuInkrementNviStatus(paNviSnvtTempP[z]^.bStatusInformation);
						EXIT;
					END_IF
				END_FOR
			END_IF
		ELSIF (cmd = M2C_NVI_UPDT_TOUT) THEN
			IF (unLastLen_mbxModule_1 = 3) THEN
				FOR z := 0 TO 8 DO
					IF aNviSnvtTempPIndex[z] = bNvRelativeIdx THEN
						paNviSnvtTempP[z]^.bStatusInformation.4 := BYTE_TO_BOOL(InDataTelegram_Module_1[2]);
						EXIT;
					END_IF
				END_FOR
			END_IF
		END_IF
	26, 32:
		IF (cmd = M2C_NVI_UPDT_OCCD) OR (cmd = M2C_NV_VALUE_RSP) THEN
			IF (unLastLen_mbxModule_1 = (2 + 2)) THEN
				FOR z := 0 TO 1 DO
					IF aNviSnvtSwitchIndex[z] = bNvRelativeIdx THEN
						FuRawToSnvtSwitch(ADR(InDataTelegram_Module_1[2]), paNviSnvtSwitch[z]);
						paNviSnvtSwitch[z]^.bInternalUseOnly.0 := FALSE;
						paNviSnvtSwitch[z]^.bStatusInformation := FuInkrementNviStatus(paNviSnvtSwitch[z]^.bStatusInformation);
						EXIT;
					END_IF
				END_FOR
			ELSIF (unLastLen_mbxModule_1 = 2) THEN
				FOR z := 0 TO 1 DO
					IF aNviSnvtSwitchIndex[z] = bNvRelativeIdx THEN
						paNviSnvtSwitch[z]^.bStatusInformation := FuInkrementNviStatus(paNviSnvtSwitch[z]^.bStatusInformation);
						EXIT;
					END_IF
				END_FOR
			END_IF
		ELSIF (cmd = M2C_NVI_UPDT_TOUT) THEN
			IF (unLastLen_mbxModule_1 = 3) THEN
				FOR z := 0 TO 1 DO
					IF aNviSnvtSwitchIndex[z] = bNvRelativeIdx THEN
						paNviSnvtSwitch[z]^.bStatusInformation.4 := BYTE_TO_BOOL(InDataTelegram_Module_1[2]);
						EXIT;
					END_IF
				END_FOR
			END_IF
		END_IF

	END_CASE
ELSIF (cmd = M2C_CP_VALUE_RSP) THEN
	wCpRelativeIdx := ((InDataTelegram_Module_1[1] + InDataTelegram_Module_1[2] * 256) - wCpStartIndex - bObjectIndex) / bLmoCount;
	CASE wCpRelativeIdx OF

	END_CASE
END_IF
END_ACTION
ACTION ResetNviUpdate:
VT_Status.bStatusInformation := VT_Status.bStatusInformation AND 16#F8;
VT_Alarm.bStatusInformation := VT_Alarm.bStatusInformation AND 16#F8;
VT_RlyState.bStatusInformation := VT_RlyState.bStatusInformation AND 16#F8;
FOR z := 0 TO 2 DO
	paNviSnvtHvacMode[z]^.bStatusInformation := paNviSnvtHvacMode[z]^.bStatusInformation AND 16#F8;
END_FOR
FOR z := 0 TO 8 DO
	paNviSnvtTempP[z]^.bStatusInformation := paNviSnvtTempP[z]^.bStatusInformation AND 16#F8;
END_FOR
FOR z := 0 TO 1 DO
	paNviSnvtSwitch[z]^.bStatusInformation := paNviSnvtSwitch[z]^.bStatusInformation AND 16#F8;
END_FOR
;
END_ACTION
ACTION SendValueRequest:
IF (FuSendNviValueReq_Module_1(ADR(VT_Status.bInternalUseOnly), bNvStartIndex + bObjectIndex + (1 * bLmoCount)) = FALSE) THEN
	RETURN;
END_IF

IF (FuSendNviValueReq_Module_1(ADR(VT_Alarm.bInternalUseOnly), bNvStartIndex + bObjectIndex + (3 * bLmoCount)) = FALSE) THEN
	RETURN;
END_IF

